LIN {X 0,Y 524.01,Z 370.549,A -85,B 0,C 180,E1 -4760.348,E2 -4760.348} C_VEL
LIN {X 0,Y 523.819,Z 378.444,A -85,B 0,C 180,E1 -4761.318,E2 -4761.318} C_VEL
LIN {X 0,Y 523.619,Z 386.151,A -85,B 0,C 180,E1 -4762.48,E2 -4762.48} C_VEL
LIN {X 0,Y 523.489,Z 393.247,A -85,B 0,C 180,E1 -4763.834,E2 -4763.834} C_VEL
LIN {X 0,Y 523.384,Z 397.968,A -85,B 0,C 180,E1 -4764.992,E2 -4764.992} C_VEL
LIN {X 0,Y 523.444,Z 401.575,A -85,B 0,C 180,E1 -4766.15,E2 -4766.15} C_VEL
LIN {X 0,Y 523.368,Z 403.434,A -85,B 0,C 180,E1 -4766.92,E2 -4766.92} C_VEL
LIN {X 0,Y 523.335,Z 404.828,A -85,B 0,C 180,E1 -4767.69,E2 -4767.69} C_VEL
LIN {X 0,Y 523.251,Z 406.428,A -85,B 0,C 180,E1 -4769.23,E2 -4769.23} C_VEL
LIN {X 0,Y 523.248,Z 406.644,A -85,B 0,C 180,E1 -4769.999,E2 -4769.999} C_VEL
LIN {X 0,Y 523.275,Z 405.822,A -85,B 0,C 180,E1 -4771.538,E2 -4771.538} C_VEL
LIN {X 0,Y 523.335,Z 404.828,A -85,B 0,C 180,E1 -4772.308,E2 -4772.308} C_VEL
LIN {X 0,Y 523.367,Z 403.433,A -85,B 0,C 180,E1 -4773.078,E2 -4773.078} C_VEL
LIN {X 0,Y 523.423,Z 400.501,A -85,B 0,C 180,E1 -4774.234,E2 -4774.234} C_VEL
LIN {X 0,Y 523.461,Z 396.528,A -85,B 0,C 180,E1 -4775.392,E2 -4775.392} C_VEL
LIN {X 0,Y 523.516,Z 391.306,A -85,B 0,C 180,E1 -4776.573,E2 -4776.573} C_VEL
LIN {X 0,Y 523.632,Z 384.971,A -85,B 0,C 180,E1 -4777.712,E2 -4777.712} C_VEL
LIN {X 0,Y 523.81,Z 376.935,A -85,B 0,C 180,E1 -4778.875,E2 -4778.875} C_VEL
LIN {X 0,Y 524.018,Z 368.739,A -85,B 0,C 180,E1 -4779.845,E2 -4779.845} C_VEL
LIN {X 0,Y 524.334,Z 358.741,A -85,B 0,C 180,E1 -4780.815,E2 -4780.815} C_VEL
LIN {X 0,Y 524.628,Z 347.427,A -85,B 0,C 180,E1 -4781.689,E2 -4781.689} C_VEL
LIN {X 0,Y 524.878,Z 336.346,A -85,B 0,C 180,E1 -4782.37,E2 -4782.37} C_VEL
LIN {X 0,Y 525.142,Z 324.039,A -85,B 0,C 180,E1 -4782.953,E2 -4782.953} C_VEL
LIN {X 0,Y 525.376,Z 311.005,A -85,B 0,C 180,E1 -4783.39,E2 -4783.39} C_VEL
LIN {X 0,Y 525.558,Z 298.573,A -85,B 0,C 180,E1 -4783.656,E2 -4783.656} C_VEL
LIN {X 0,Y 525.847,Z 204.835,A -85,B 0,C 180,E1 -4784.959,E2 -4784.959} C_VEL
LIN {X 0,Y 524.268,Z 194.811,A -85,B 0,C 180,E1 -4785.162,E2 -4785.162} C_VEL
LIN {X 0,Y 524.289,Z 192.055,A -85,B 0,C 180,E1 -4785.55,E2 -4785.55} C_VEL
LIN {X 0,Y 524.689,Z 173.78,A -85,B 0,C 180,E1 -4788.528,E2 -4788.528} C_VEL
LIN {X 0,Y 525.146,Z 153.996,A -85,B 0,C 180,E1 -4791.799,E2 -4791.799} C_VEL
LIN {X 0,Y 524.744,Z 149.225,A -85,B 0,C 180,E1 -4792.618,E2 -4792.618} C_VEL
LIN {X 0,Y 523.947,Z 144.887,A -85,B 0,C 180,E1 -4793.413,E2 -4793.413} C_VEL
LIN {X 0,Y 523.895,Z 144.725,A -85,B 0,C 180,E1 -4796.274,E2 -4796.274} C_VEL
LIN {X 0,Y 523.867,Z 144.728,A -85,B 0,C 180,E1 -4798.878,E2 -4798.878} C_VEL
LIN {X 0,Y 523.903,Z 144.728,A -85,B 0,C 180,E1 -4801.544,E2 -4801.544} C_VEL
LIN {X 0,Y 523.906,Z 144.722,A -85,B 0,C 180,E1 -4804.291,E2 -4804.291} C_VEL
LIN {X 0,Y 523.861,Z 144.732,A -85,B 0,C 180,E1 -4807.671,E2 -4807.671} C_VEL
LIN {X 0,Y 523.906,Z 144.721,A -85,B 0,C 180,E1 -4810.125,E2 -4810.125} C_VEL
LIN {X 0,Y 523.864,Z 144.732,A -85,B 0,C 180,E1 -4813.171,E2 -4813.171} C_VEL
LIN {X 0,Y 523.909,Z 144.723,A -85,B 0,C 180,E1 -4815.768,E2 -4815.768} C_VEL
LIN {X 0,Y 523.882,Z 144.728,A -85,B 0,C 180,E1 -4818.902,E2 -4818.902} C_VEL
LIN {X 0,Y 523.891,Z 144.722,A -85,B 0,C 180,E1 -4821.896,E2 -4821.896} C_VEL
LIN {X 0,Y 523.907,Z 144.726,A -85,B 0,C 180,E1 -4824.911,E2 -4824.911} C_VEL
LIN {X 0,Y 523.889,Z 144.724,A -85,B 0,C 180,E1 -4827.685,E2 -4827.685} C_VEL
LIN {X 0,Y 523.919,Z 144.722,A -85,B 0,C 180,E1 -4830.68,E2 -4830.68} C_VEL
LIN {X 0,Y 523.888,Z 144.723,A -85,B 0,C 180,E1 -4833.724,E2 -4833.724} C_VEL
LIN {X 0,Y 523.894,Z 144.722,A -85,B 0,C 180,E1 -4836.268,E2 -4836.268} C_VEL
LIN {X 0,Y 523.929,Z 144.724,A -85,B 0,C 180,E1 -4838.766,E2 -4838.766} C_VEL
LIN {X 0,Y 523.918,Z 144.722,A -85,B 0,C 180,E1 -4841.219,E2 -4841.219} C_VEL
LIN {X 0,Y 523.894,Z 144.721,A -85,B 0,C 180,E1 -4843.637,E2 -4843.637} C_VEL
LIN {X 0,Y 523.897,Z 144.721,A -85,B 0,C 180,E1 -4846.026,E2 -4846.026} C_VEL
LIN {X 0,Y 524,Z 144.712,A -85,B 0,C 180,E1 -4848.393,E2 -4848.393} C_VEL
LIN {X 0,Y 523.967,Z 144.713,A -85,B 0,C 180,E1 -4851.515,E2 -4851.515} C_VEL
LIN {X 0,Y 523.999,Z 144.708,A -85,B 0,C 180,E1 -4853.84,E2 -4853.84} C_VEL
LIN {X 0,Y 524.02,Z 144.71,A -85,B 0,C 180,E1 -4856.924,E2 -4856.924} C_VEL
LIN {X 0,Y 523.982,Z 144.718,A -85,B 0,C 180,E1 -4858.462,E2 -4858.462} C_VEL
LIN {X 0,Y 524.105,Z 144.702,A -85,B 0,C 180,E1 -4860.768,E2 -4860.768} C_VEL
LIN {X 0,Y 524.011,Z 144.707,A -85,B 0,C 180,E1 -4863.075,E2 -4863.075} C_VEL
LIN {X 0,Y 523.998,Z 144.714,A -85,B 0,C 180,E1 -4866.159,E2 -4866.159} C_VEL
LIN {X 0,Y 523.959,Z 144.713,A -85,B 0,C 180,E1 -4869.262,E2 -4869.262} C_VEL
LIN {X 0,Y 523.937,Z 144.725,A -85,B 0,C 180,E1 -4872.393,E2 -4872.393} C_VEL
LIN {X 0,Y 523.907,Z 144.721,A -85,B 0,C 180,E1 -4875.562,E2 -4875.562} C_VEL
LIN {X 0,Y 523.9,Z 144.727,A -85,B 0,C 180,E1 -4877.971,E2 -4877.971} C_VEL
LIN {X 0,Y 523.957,Z 144.721,A -85,B 0,C 180,E1 -4880.41,E2 -4880.41} C_VEL
LIN {X 0,Y 523.894,Z 144.724,A -85,B 0,C 180,E1 -4882.894,E2 -4882.894} C_VEL
LIN {X 0,Y 523.883,Z 144.724,A -85,B 0,C 180,E1 -4885.422,E2 -4885.422} C_VEL
LIN {X 0,Y 523.882,Z 144.732,A -85,B 0,C 180,E1 -4888.004,E2 -4888.004} C_VEL
LIN {X 0,Y 523.917,Z 144.724,A -85,B 0,C 180,E1 -4890.852,E2 -4890.852} C_VEL
LIN {X 0,Y 523.983,Z 144.932,A -85,B 0,C 180,E1 -4892.759,E2 -4892.759} C_VEL
LIN {X 0,Y 524.746,Z 150.857,A -85,B 0,C 180,E1 -4893.865,E2 -4893.865} C_VEL
LIN {X 0,Y 524.446,Z 167.206,A -85,B 0,C 180,E1 -4896.753,E2 -4896.753} C_VEL
LIN {X 0,Y 524.249,Z 179.439,A -85,B 0,C 180,E1 -4898.871,E2 -4898.871} C_VEL
LIN {X 0,Y 525.481,Z 186.461,A -85,B 0,C 180,E1 -4899.038,E2 -4899.038} C_VEL
LIN {X 0,Y 525.936,Z 190.572,A -85,B 0,C 180,E1 -4899.109,E2 -4899.109} C_VEL
LIN {X 0,Y 525.754,Z 232.261,A -85,B 0,C 180,E1 -4899.688,E2 -4899.688} C_VEL
LIN {X 0,Y 524.994,Z 238.101,A -85,B 0,C 180,E1 -4899.748,E2 -4899.748} C_VEL
LIN {X 0,Y 519.456,Z 257.107,A -85,B 0,C 180,E1 -4899.861,E2 -4899.861} C_VEL
LIN {X 0,Y 518.757,Z 262.947,A -85,B 0,C 180,E1 -4899.924,E2 -4899.924} C_VEL
LIN {X 0,Y 518.573,Z 288.396,A -85,B 0,C 180,E1 -4900.31,E2 -4900.31} C_VEL
LIN {X 0,Y 518.38,Z 301.986,A -85,B 0,C 180,E1 -4900.685,E2 -4900.685} C_VEL
LIN {X 0,Y 518.137,Z 314.524,A -85,B 0,C 180,E1 -4901.2,E2 -4901.2} C_VEL
LIN {X 0,Y 517.792,Z 326.753,A -85,B 0,C 180,E1 -4901.876,E2 -4901.876} C_VEL
LIN {X 0,Y 517.482,Z 338.316,A -85,B 0,C 180,E1 -4902.703,E2 -4902.703} C_VEL
LIN {X 0,Y 517.193,Z 348.83,A -85,B 0,C 180,E1 -4903.65,E2 -4903.65} C_VEL
LIN {X 0,Y 516.919,Z 358.553,A -85,B 0,C 180,E1 -4904.736,E2 -4904.736} C_VEL
LIN {X 0,Y 516.679,Z 366.293,A -85,B 0,C 180,E1 -4905.806,E2 -4905.806} C_VEL
LIN {X 0,Y 516.532,Z 372.681,A -85,B 0,C 180,E1 -4906.883,E2 -4906.883} C_VEL
LIN {X 0,Y 516.407,Z 378.822,A -85,B 0,C 180,E1 -4908.177,E2 -4908.177} C_VEL
LIN {X 0,Y 516.331,Z 384.126,A -85,B 0,C 180,E1 -4909.661,E2 -4909.661} C_VEL
LIN {X 0,Y 516.176,Z 387.85,A -85,B 0,C 180,E1 -4911.223,E2 -4911.223} C_VEL
LIN {X 0,Y 516.139,Z 389.373,A -85,B 0,C 180,E1 -4912.214,E2 -4912.214} C_VEL
LIN {X 0,Y 516.127,Z 390.348,A -85,B 0,C 180,E1 -4913.455,E2 -4913.455} C_VEL
LIN {X 0,Y 516.161,Z 390.29,A -85,B 0,C 180,E1 -4914.78,E2 -4914.78} C_VEL
LIN {X 0,Y 516.171,Z 389.02,A -85,B 0,C 180,E1 -4916.155,E2 -4916.155} C_VEL
LIN {X 0,Y 516.28,Z 386.4,A -85,B 0,C 180,E1 -4917.563,E2 -4917.563} C_VEL
LIN {X 0,Y 516.323,Z 382.764,A -85,B 0,C 180,E1 -4918.854,E2 -4918.854} C_VEL
LIN {X 0,Y 516.43,Z 377.59,A -85,B 0,C 180,E1 -4920.195,E2 -4920.195} C_VEL
LIN {X 0,Y 516.542,Z 371.937,A -85,B 0,C 180,E1 -4921.342,E2 -4921.342} C_VEL
LIN {X 0,Y 516.768,Z 363.589,A -85,B 0,C 180,E1 -4922.679,E2 -4922.679} C_VEL
LIN {X 0,Y 517.007,Z 354.868,A -85,B 0,C 180,E1 -4923.789,E2 -4923.789} C_VEL
LIN {X 0,Y 517.288,Z 345.382,A -85,B 0,C 180,E1 -4924.77,E2 -4924.77} C_VEL
LIN {X 0,Y 517.613,Z 334.613,A -85,B 0,C 180,E1 -4925.671,E2 -4925.671} C_VEL
LIN {X 0,Y 517.889,Z 323.665,A -85,B 0,C 180,E1 -4926.403,E2 -4926.403} C_VEL
LIN {X 0,Y 518.19,Z 311.591,A -85,B 0,C 180,E1 -4927.023,E2 -4927.023} C_VEL
LIN {X 0,Y 518.39,Z 298.873,A -85,B 0,C 180,E1 -4927.507,E2 -4927.507} C_VEL
LIN {X 0,Y 518.613,Z 285.867,A -85,B 0,C 180,E1 -4927.833,E2 -4927.833} C_VEL
LIN {X 0,Y 519.067,Z 189.85,A -85,B 0,C 180,E1 -4929.195,E2 -4929.195} C_VEL
LIN {X 0,Y 517.279,Z 179.688,A -85,B 0,C 180,E1 -4929.42,E2 -4929.42} C_VEL
LIN {X 0,Y 517.451,Z 169.81,A -85,B 0,C 180,E1 -4931.183,E2 -4931.183} C_VEL
LIN {X 0,Y 517.932,Z 153.223,A -85,B 0,C 180,E1 -4934.254,E2 -4934.254} C_VEL
LIN {X 0,Y 517.574,Z 149.071,A -85,B 0,C 180,E1 -4935.05,E2 -4935.05} C_VEL
LIN {X 0,Y 516.951,Z 145.624,A -85,B 0,C 180,E1 -4935.786,E2 -4935.786} C_VEL
LIN {X 0,Y 516.948,Z 145.59,A -85,B 0,C 180,E1 -4939.029,E2 -4939.029} C_VEL
LIN {X 0,Y 516.975,Z 145.588,A -85,B 0,C 180,E1 -4942.188,E2 -4942.188} C_VEL
LIN {X 0,Y 517.026,Z 145.578,A -85,B 0,C 180,E1 -4944.541,E2 -4944.541} C_VEL
LIN {X 0,Y 517.08,Z 145.577,A -85,B 0,C 180,E1 -4947.664,E2 -4947.664} C_VEL
LIN {X 0,Y 517.091,Z 145.569,A -85,B 0,C 180,E1 -4950.78,E2 -4950.78} C_VEL
LIN {X 0,Y 517.01,Z 145.581,A -85,B 0,C 180,E1 -4953.118,E2 -4953.118} C_VEL
LIN {X 0,Y 517,Z 145.581,A -85,B 0,C 180,E1 -4956.244,E2 -4956.244} C_VEL
LIN {X 0,Y 516.946,Z 145.594,A -85,B 0,C 180,E1 -4959.39,E2 -4959.39} C_VEL
LIN {X 0,Y 516.95,Z 145.591,A -85,B 0,C 180,E1 -4961.808,E2 -4961.808} C_VEL
LIN {X 0,Y 516.943,Z 145.592,A -85,B 0,C 180,E1 -4965.147,E2 -4965.147} C_VEL
LIN {X 0,Y 516.915,Z 145.591,A -85,B 0,C 180,E1 -4968.223,E2 -4968.223} C_VEL
LIN {X 0,Y 516.911,Z 145.593,A -85,B 0,C 180,E1 -4970.702,E2 -4970.702} C_VEL
LIN {X 0,Y 516.889,Z 145.594,A -85,B 0,C 180,E1 -4974.074,E2 -4974.074} C_VEL
LIN {X 0,Y 516.923,Z 145.592,A -85,B 0,C 180,E1 -4976.658,E2 -4976.658} C_VEL
LIN {X 0,Y 516.908,Z 145.595,A -85,B 0,C 180,E1 -4979.524,E2 -4979.524} C_VEL
LIN {X 0,Y 516.893,Z 145.596,A -85,B 0,C 180,E1 -4982.543,E2 -4982.543} C_VEL
LIN {X 0,Y 516.864,Z 145.601,A -85,B 0,C 180,E1 -4985.33,E2 -4985.33} C_VEL
LIN {X 0,Y 516.878,Z 145.595,A -85,B 0,C 180,E1 -4987.943,E2 -4987.943} C_VEL
LIN {X 0,Y 516.882,Z 145.602,A -85,B 0,C 180,E1 -4990.742,E2 -4990.742} C_VEL
LIN {X 0,Y 516.881,Z 145.604,A -85,B 0,C 180,E1 -4992.832,E2 -4992.832} C_VEL
LIN {X 0,Y 516.894,Z 145.599,A -85,B 0,C 180,E1 -4995.007,E2 -4995.007} C_VEL
LIN {X 0,Y 516.908,Z 145.596,A -85,B 0,C 180,E1 -4998.4,E2 -4998.4} C_VEL
LIN {X 0,Y 516.877,Z 145.596,A -85,B 0,C 180,E1 -5001.284,E2 -5001.284} C_VEL
LIN {X 0,Y 516.866,Z 145.601,A -85,B 0,C 180,E1 -5004.22,E2 -5004.22} C_VEL
LIN {X 0,Y 516.893,Z 145.595,A -85,B 0,C 180,E1 -5007.053,E2 -5007.053} C_VEL
LIN {X 0,Y 516.886,Z 145.596,A -85,B 0,C 180,E1 -5009.796,E2 -5009.796} C_VEL
LIN {X 0,Y 516.891,Z 145.602,A -85,B 0,C 180,E1 -5012.466,E2 -5012.466} C_VEL
LIN {X 0,Y 516.864,Z 145.598,A -85,B 0,C 180,E1 -5015.07,E2 -5015.07} C_VEL
LIN {X 0,Y 516.868,Z 145.598,A -85,B 0,C 180,E1 -5017.622,E2 -5017.622} C_VEL
LIN {X 0,Y 516.928,Z 145.597,A -85,B 0,C 180,E1 -5020.13,E2 -5020.13} C_VEL
LIN {X 0,Y 516.892,Z 145.597,A -85,B 0,C 180,E1 -5022.595,E2 -5022.595} C_VEL
LIN {X 0,Y 516.934,Z 145.588,A -85,B 0,C 180,E1 -5025.03,E2 -5025.03} C_VEL
LIN {X 0,Y 516.966,Z 145.59,A -85,B 0,C 180,E1 -5028.234,E2 -5028.234} C_VEL
LIN {X 0,Y 516.934,Z 145.59,A -85,B 0,C 180,E1 -5031.399,E2 -5031.399} C_VEL
LIN {X 0,Y 516.985,Z 145.583,A -85,B 0,C 180,E1 -5034.54,E2 -5034.54} C_VEL
LIN {X 0,Y 517.072,Z 145.578,A -85,B 0,C 180,E1 -5037.663,E2 -5037.663} C_VEL
LIN {X 0,Y 517.063,Z 145.578,A -85,B 0,C 180,E1 -5040,E2 -5040} C_VEL
LIN {X 0,Y 517.073,Z 145.572,A -85,B 0,C 180,E1 -5042.337,E2 -5042.337} C_VEL
LIN {X 0,Y 516.98,Z 145.589,A -85,B 0,C 180,E1 -5045.461,E2 -5045.461} C_VEL
LIN {X 0,Y 516.926,Z 145.589,A -85,B 0,C 180,E1 -5048.601,E2 -5048.601} C_VEL
LIN {X 0,Y 516.953,Z 145.591,A -85,B 0,C 180,E1 -5051.807,E2 -5051.807} C_VEL
LIN {X 0,Y 516.935,Z 145.593,A -85,B 0,C 180,E1 -5055.142,E2 -5055.142} C_VEL
LIN {X 0,Y 516.876,Z 145.596,A -85,B 0,C 180,E1 -5058.224,E2 -5058.224} C_VEL
LIN {X 0,Y 516.894,Z 145.595,A -85,B 0,C 180,E1 -5060.703,E2 -5060.703} C_VEL
LIN {X 0,Y 516.856,Z 145.606,A -85,B 0,C 180,E1 -5063.225,E2 -5063.225} C_VEL
LIN {X 0,Y 516.86,Z 145.598,A -85,B 0,C 180,E1 -5066.177,E2 -5066.177} C_VEL
LIN {X 0,Y 516.829,Z 145.602,A -85,B 0,C 180,E1 -5068.421,E2 -5068.421} C_VEL
LIN {X 0,Y 516.849,Z 145.608,A -85,B 0,C 180,E1 -5071.113,E2 -5071.113} C_VEL
LIN {X 0,Y 516.871,Z 145.596,A -85,B 0,C 180,E1 -5073.96,E2 -5073.96} C_VEL
LIN {X 0,Y 516.81,Z 145.609,A -85,B 0,C 180,E1 -5076.752,E2 -5076.752} C_VEL
LIN {X 0,Y 516.866,Z 145.602,A -85,B 0,C 180,E1 -5079.19,E2 -5079.19} C_VEL
LIN {X 0,Y 516.832,Z 145.601,A -85,B 0,C 180,E1 -5081.784,E2 -5081.784} C_VEL
LIN {X 0,Y 516.898,Z 145.599,A -85,B 0,C 180,E1 -5085.007,E2 -5085.007} C_VEL
LIN {X 0,Y 516.831,Z 145.605,A -85,B 0,C 180,E1 -5088.41,E2 -5088.41} C_VEL
LIN {X 0,Y 516.85,Z 145.6,A -85,B 0,C 180,E1 -5091.281,E2 -5091.281} C_VEL
LIN {X 0,Y 516.809,Z 145.612,A -85,B 0,C 180,E1 -5094.68,E2 -5094.68} C_VEL
LIN {X 0,Y 516.865,Z 145.597,A -85,B 0,C 180,E1 -5097.463,E2 -5097.463} C_VEL
LIN {X 0,Y 516.84,Z 145.609,A -85,B 0,C 180,E1 -5100.491,E2 -5100.491} C_VEL
LIN {X 0,Y 516.831,Z 145.602,A -85,B 0,C 180,E1 -5103.337,E2 -5103.337} C_VEL
LIN {X 0,Y 516.911,Z 145.72,A -85,B 0,C 180,E1 -5106.3,E2 -5106.3} C_VEL
LIN {X 0,Y 518.219,Z 153.145,A -85,B 0,C 180,E1 -5107.682,E2 -5107.682} C_VEL
LIN {X 0,Y 517.907,Z 166.623,A -85,B 0,C 180,E1 -5109.977,E2 -5109.977} C_VEL
LIN {X 0,Y 517.502,Z 183.566,A -85,B 0,C 180,E1 -5112.819,E2 -5112.819} C_VEL
LIN {X 0,Y 517.266,Z 194.642,A -85,B 0,C 180,E1 -5114.617,E2 -5114.617} C_VEL
LIN {X 0,Y 519.088,Z 206.76,A -85,B 0,C 180,E1 -5114.869,E2 -5114.869} C_VEL
LIN {X 0,Y 518.62,Z 302.588,A -85,B 0,C 180,E1 -5116.231,E2 -5116.231} C_VEL
LIN {X 0,Y 518.394,Z 315.759,A -85,B 0,C 180,E1 -5116.575,E2 -5116.575} C_VEL
LIN {X 0,Y 518.099,Z 328.438,A -85,B 0,C 180,E1 -5117.066,E2 -5117.066} C_VEL
LIN {X 0,Y 517.853,Z 339.954,A -85,B 0,C 180,E1 -5117.672,E2 -5117.672} C_VEL
LIN {X 0,Y 517.56,Z 351.366,A -85,B 0,C 180,E1 -5118.445,E2 -5118.445} C_VEL
LIN {X 0,Y 517.223,Z 361.847,A -85,B 0,C 180,E1 -5119.33,E2 -5119.33} C_VEL
LIN {X 0,Y 516.955,Z 370.414,A -85,B 0,C 180,E1 -5120.215,E2 -5120.215} C_VEL
LIN {X 0,Y 516.756,Z 378.314,A -85,B 0,C 180,E1 -5121.198,E2 -5121.198} C_VEL
LIN {X 0,Y 516.545,Z 386.028,A -85,B 0,C 180,E1 -5122.376,E2 -5122.376} C_VEL
LIN {X 0,Y 516.399,Z 393.129,A -85,B 0,C 180,E1 -5123.749,E2 -5123.749} C_VEL
LIN {X 0,Y 516.313,Z 397.852,A -85,B 0,C 180,E1 -5124.923,E2 -5124.923} C_VEL
LIN {X 0,Y 516.352,Z 401.462,A -85,B 0,C 180,E1 -5126.097,E2 -5126.097} C_VEL
LIN {X 0,Y 516.283,Z 403.323,A -85,B 0,C 180,E1 -5126.878,E2 -5126.878} C_VEL
LIN {X 0,Y 516.262,Z 404.718,A -85,B 0,C 180,E1 -5127.659,E2 -5127.659} C_VEL
LIN {X 0,Y 516.16,Z 406.318,A -85,B 0,C 180,E1 -5129.219,E2 -5129.219} C_VEL
LIN {X 0,Y 516.156,Z 406.534,A -85,B 0,C 180,E1 -5129.999,E2 -5129.999} C_VEL
LIN {X 0,Y 516.192,Z 405.711,A -85,B 0,C 180,E1 -5131.56,E2 -5131.56} C_VEL
LIN {X 0,Y 516.261,Z 404.716,A -85,B 0,C 180,E1 -5132.34,E2 -5132.34} C_VEL
LIN {X 0,Y 516.282,Z 403.319,A -85,B 0,C 180,E1 -5133.12,E2 -5133.12} C_VEL
LIN {X 0,Y 516.311,Z 400.383,A -85,B 0,C 180,E1 -5134.293,E2 -5134.293} C_VEL
LIN {X 0,Y 516.397,Z 396.408,A -85,B 0,C 180,E1 -5135.466,E2 -5135.466} C_VEL
LIN {X 0,Y 516.48,Z 390.481,A -85,B 0,C 180,E1 -5136.8,E2 -5136.8} C_VEL
LIN {X 0,Y 516.586,Z 383.604,A -85,B 0,C 180,E1 -5138.015,E2 -5138.015} C_VEL
LIN {X 0,Y 516.806,Z 375.304,A -85,B 0,C 180,E1 -5139.194,E2 -5139.194} C_VEL
LIN {X 0,Y 517.027,Z 366.785,A -85,B 0,C 180,E1 -5140.177,E2 -5140.177} C_VEL
LIN {X 0,Y 517.375,Z 356.259,A -85,B 0,C 180,E1 -5141.16,E2 -5141.16} C_VEL
LIN {X 0,Y 517.707,Z 344.792,A -85,B 0,C 180,E1 -5142.019,E2 -5142.019} C_VEL
LIN {X 0,Y 517.987,Z 334.391,A -85,B 0,C 180,E1 -5142.636,E2 -5142.636} C_VEL
LIN {X 0,Y 518.243,Z 322.571,A -85,B 0,C 180,E1 -5143.178,E2 -5143.178} C_VEL
LIN {X 0,Y 518.494,Z 308.936,A -85,B 0,C 180,E1 -5143.621,E2 -5143.621} C_VEL
LIN {X 0,Y 518.668,Z 295.053,A -85,B 0,C 180,E1 -5143.891,E2 -5143.891} C_VEL
LIN {X 0,Y 518.972,Z 205.308,A -85,B 0,C 180,E1 -5145.153,E2 -5145.153} C_VEL
LIN {X 0,Y 517.263,Z 194.623,A -85,B 0,C 180,E1 -5145.375,E2 -5145.375} C_VEL
LIN {X 0,Y 517.4,Z 187.023,A -85,B 0,C 180,E1 -5146.573,E2 -5146.573} C_VEL
LIN {X 0,Y 517.776,Z 169.838,A -85,B 0,C 180,E1 -5149.422,E2 -5149.422} C_VEL
LIN {X 0,Y 518.209,Z 153.859,A -85,B 0,C 180,E1 -5152.106,E2 -5152.106} C_VEL
LIN {X 0,Y 516.916,Z 145.723,A -85,B 0,C 180,E1 -5153.591,E2 -5153.591} C_VEL
LIN {X 0,Y 516.833,Z 145.604,A -85,B 0,C 180,E1 -5156.662,E2 -5156.662} C_VEL
LIN {X 0,Y 516.834,Z 145.608,A -85,B 0,C 180,E1 -5159.508,E2 -5159.508} C_VEL
LIN {X 0,Y 516.887,Z 145.596,A -85,B 0,C 180,E1 -5162.541,E2 -5162.541} C_VEL
LIN {X 0,Y 516.844,Z 145.608,A -85,B 0,C 180,E1 -5165.326,E2 -5165.326} C_VEL
LIN {X 0,Y 516.851,Z 145.6,A -85,B 0,C 180,E1 -5168.717,E2 -5168.717} C_VEL
LIN {X 0,Y 516.834,Z 145.605,A -85,B 0,C 180,E1 -5171.781,E2 -5171.781} C_VEL
LIN {X 0,Y 516.888,Z 145.599,A -85,B 0,C 180,E1 -5175.006,E2 -5175.006} C_VEL
LIN {X 0,Y 516.841,Z 145.601,A -85,B 0,C 180,E1 -5178.406,E2 -5178.406} C_VEL
LIN {X 0,Y 516.861,Z 145.605,A -85,B 0,C 180,E1 -5181.282,E2 -5181.282} C_VEL
LIN {X 0,Y 516.849,Z 145.602,A -85,B 0,C 180,E1 -5184.67,E2 -5184.67} C_VEL
LIN {X 0,Y 516.856,Z 145.602,A -85,B 0,C 180,E1 -5187.461,E2 -5187.461} C_VEL
LIN {X 0,Y 516.887,Z 145.598,A -85,B 0,C 180,E1 -5190.693,E2 -5190.693} C_VEL
LIN {X 0,Y 516.868,Z 145.597,A -85,B 0,C 180,E1 -5193.817,E2 -5193.817} C_VEL
LIN {X 0,Y 516.843,Z 145.605,A -85,B 0,C 180,E1 -5196.775,E2 -5196.775} C_VEL
LIN {X 0,Y 516.917,Z 145.59,A -85,B 0,C 180,E1 -5199.734,E2 -5199.734} C_VEL
LIN {X 0,Y 516.88,Z 145.6,A -85,B 0,C 180,E1 -5202.594,E2 -5202.594} C_VEL
LIN {X 0,Y 516.916,Z 145.596,A -85,B 0,C 180,E1 -5205.029,E2 -5205.029} C_VEL
LIN {X 0,Y 516.953,Z 145.588,A -85,B 0,C 180,E1 -5208.233,E2 -5208.233} C_VEL
LIN {X 0,Y 516.935,Z 145.589,A -85,B 0,C 180,E1 -5211.399,E2 -5211.399} C_VEL
LIN {X 0,Y 516.968,Z 145.584,A -85,B 0,C 180,E1 -5213.756,E2 -5213.756} C_VEL
LIN {X 0,Y 516.963,Z 145.59,A -85,B 0,C 180,E1 -5216.882,E2 -5216.882} C_VEL
LIN {X 0,Y 516.95,Z 145.593,A -85,B 0,C 180,E1 -5218.442,E2 -5218.442} C_VEL
LIN {X 0,Y 517.075,Z 145.577,A -85,B 0,C 180,E1 -5220.778,E2 -5220.778} C_VEL
LIN {X 0,Y 516.952,Z 145.586,A -85,B 0,C 180,E1 -5223.117,E2 -5223.117} C_VEL
LIN {X 0,Y 516.967,Z 145.591,A -85,B 0,C 180,E1 -5226.243,E2 -5226.243} C_VEL
LIN {X 0,Y 516.914,Z 145.591,A -85,B 0,C 180,E1 -5229.39,E2 -5229.39} C_VEL
LIN {X 0,Y 516.889,Z 145.601,A -85,B 0,C 180,E1 -5232.565,E2 -5232.565} C_VEL
LIN {X 0,Y 516.928,Z 145.59,A -85,B 0,C 180,E1 -5235.145,E2 -5235.145} C_VEL
LIN {X 0,Y 516.862,Z 145.606,A -85,B 0,C 180,E1 -5238.224,E2 -5238.224} C_VEL
LIN {X 0,Y 516.897,Z 145.597,A -85,B 0,C 180,E1 -5240.702,E2 -5240.702} C_VEL
LIN {X 0,Y 516.87,Z 145.605,A -85,B 0,C 180,E1 -5244.074,E2 -5244.074} C_VEL
LIN {X 0,Y 516.822,Z 145.606,A -85,B 0,C 180,E1 -5246.663,E2 -5246.663} C_VEL
LIN {X 0,Y 516.87,Z 145.602,A -85,B 0,C 180,E1 -5249.519,E2 -5249.519} C_VEL
LIN {X 0,Y 516.937,Z 145.733,A -85,B 0,C 180,E1 -5252.593,E2 -5252.593} C_VEL
LIN {X 0,Y 517.785,Z 152.112,A -85,B 0,C 180,E1 -5253.814,E2 -5253.814} C_VEL
LIN {X 0,Y 517.435,Z 169.647,A -85,B 0,C 180,E1 -5256.942,E2 -5256.942} C_VEL
LIN {X 0,Y 517.285,Z 179.482,A -85,B 0,C 180,E1 -5258.656,E2 -5258.656} C_VEL
LIN {X 0,Y 518.114,Z 184.368,A -85,B 0,C 180,E1 -5258.788,E2 -5258.788} C_VEL
LIN {X 0,Y 519.099,Z 190.699,A -85,B 0,C 180,E1 -5258.908,E2 -5258.908} C_VEL
LIN {X 0,Y 518.757,Z 262.947,A -85,B 0,C 180,E1 -5259.924,E2 -5259.924} C_VEL
LIN {X 0,Y 518.026,Z 268.8,A -85,B 0,C 180,E1 -5259.982,E2 -5259.982} C_VEL
LIN {X 0,Y 512.332,Z 287.754,A -85,B 0,C 180,E1 -5260.122,E2 -5260.122} C_VEL
LIN {X 0,Y 511.653,Z 293.501,A -85,B 0,C 180,E1 -5260.244,E2 -5260.244} C_VEL
LIN {X 0,Y 511.389,Z 306.53,A -85,B 0,C 180,E1 -5260.67,E2 -5260.67} C_VEL
LIN {X 0,Y 511.121,Z 318.867,A -85,B 0,C 180,E1 -5261.241,E2 -5261.241} C_VEL
LIN {X 0,Y 510.819,Z 330.246,A -85,B 0,C 180,E1 -5261.938,E2 -5261.938} C_VEL
LIN {X 0,Y 510.423,Z 341.048,A -85,B 0,C 180,E1 -5262.77,E2 -5262.77} C_VEL
LIN {X 0,Y 510.143,Z 350.656,A -85,B 0,C 180,E1 -5263.685,E2 -5263.685} C_VEL
LIN {X 0,Y 509.87,Z 359.112,A -85,B 0,C 180,E1 -5264.666,E2 -5264.666} C_VEL
LIN {X 0,Y 509.625,Z 367.176,A -85,B 0,C 180,E1 -5265.816,E2 -5265.816} C_VEL
LIN {X 0,Y 509.456,Z 373.805,A -85,B 0,C 180,E1 -5266.981,E2 -5266.981} C_VEL
LIN {X 0,Y 509.332,Z 379.223,A -85,B 0,C 180,E1 -5268.169,E2 -5268.169} C_VEL
LIN {X 0,Y 509.247,Z 384.12,A -85,B 0,C 180,E1 -5269.563,E2 -5269.563} C_VEL
LIN {X 0,Y 509.148,Z 386.847,A -85,B 0,C 180,E1 -5270.623,E2 -5270.623} C_VEL
LIN {X 0,Y 509.056,Z 389.128,A -85,B 0,C 180,E1 -5271.9,E2 -5271.9} C_VEL
LIN {X 0,Y 509.029,Z 390.362,A -85,B 0,C 180,E1 -5273.205,E2 -5273.205} C_VEL
LIN {X 0,Y 509.047,Z 390.497,A -85,B 0,C 180,E1 -5274.561,E2 -5274.561} C_VEL
LIN {X 0,Y 509.067,Z 389.454,A -85,B 0,C 180,E1 -5275.928,E2 -5275.928} C_VEL
LIN {X 0,Y 509.169,Z 386.907,A -85,B 0,C 180,E1 -5277.433,E2 -5277.433} C_VEL
LIN {X 0,Y 509.228,Z 383.142,A -85,B 0,C 180,E1 -5278.834,E2 -5278.834} C_VEL
LIN {X 0,Y 509.362,Z 377.969,A -85,B 0,C 180,E1 -5280.219,E2 -5280.219} C_VEL
LIN {X 0,Y 509.497,Z 371.257,A -85,B 0,C 180,E1 -5281.582,E2 -5281.582} C_VEL
LIN {X 0,Y 509.725,Z 364.247,A -85,B 0,C 180,E1 -5282.715,E2 -5282.715} C_VEL
LIN {X 0,Y 509.974,Z 355.742,A -85,B 0,C 180,E1 -5283.834,E2 -5283.834} C_VEL
LIN {X 0,Y 510.28,Z 345.716,A -85,B 0,C 180,E1 -5284.895,E2 -5284.895} C_VEL
LIN {X 0,Y 510.639,Z 334.687,A -85,B 0,C 180,E1 -5285.831,E2 -5285.831} C_VEL
LIN {X 0,Y 510.972,Z 323.625,A -85,B 0,C 180,E1 -5286.578,E2 -5286.578} C_VEL
LIN {X 0,Y 511.269,Z 311.047,A -85,B 0,C 180,E1 -5287.229,E2 -5287.229} C_VEL
LIN {X 0,Y 511.571,Z 297.863,A -85,B 0,C 180,E1 -5287.724,E2 -5287.724} C_VEL
LIN {X 0,Y 511.741,Z 285.725,A -85,B 0,C 180,E1 -5288.024,E2 -5288.024} C_VEL
LIN {X 0,Y 512.111,Z 189.928,A -85,B 0,C 180,E1 -5289.405,E2 -5289.405} C_VEL
LIN {X 0,Y 510.291,Z 179.816,A -85,B 0,C 180,E1 -5289.632,E2 -5289.632} C_VEL
LIN {X 0,Y 510.408,Z 173.744,A -85,B 0,C 180,E1 -5290.704,E2 -5290.704} C_VEL
LIN {X 0,Y 510.931,Z 155.967,A -85,B 0,C 180,E1 -5294.033,E2 -5294.033} C_VEL
LIN {X 0,Y 510.67,Z 150.691,A -85,B 0,C 180,E1 -5295.047,E2 -5295.047} C_VEL
LIN {X 0,Y 509.889,Z 146.503,A -85,B 0,C 180,E1 -5295.941,E2 -5295.941} C_VEL
LIN {X 0,Y 509.91,Z 146.467,A -85,B 0,C 180,E1 -5298.875,E2 -5298.875} C_VEL
LIN {X 0,Y 509.949,Z 146.465,A -85,B 0,C 180,E1 -5302.079,E2 -5302.079} C_VEL
LIN {X 0,Y 509.978,Z 146.456,A -85,B 0,C 180,E1 -5304.465,E2 -5304.465} C_VEL
LIN {X 0,Y 510.051,Z 146.452,A -85,B 0,C 180,E1 -5307.632,E2 -5307.632} C_VEL
LIN {X 0,Y 510.061,Z 146.445,A -85,B 0,C 180,E1 -5310.79,E2 -5310.79} C_VEL
LIN {X 0,Y 509.952,Z 146.46,A -85,B 0,C 180,E1 -5313.161,E2 -5313.161} C_VEL
LIN {X 0,Y 509.952,Z 146.459,A -85,B 0,C 180,E1 -5316.331,E2 -5316.331} C_VEL
LIN {X 0,Y 509.888,Z 146.475,A -85,B 0,C 180,E1 -5319.521,E2 -5319.521} C_VEL
LIN {X 0,Y 509.903,Z 146.467,A -85,B 0,C 180,E1 -5321.932,E2 -5321.932} C_VEL
LIN {X 0,Y 509.893,Z 146.472,A -85,B 0,C 180,E1 -5325.242,E2 -5325.242} C_VEL
LIN {X 0,Y 509.86,Z 146.47,A -85,B 0,C 180,E1 -5328.484,E2 -5328.484} C_VEL
LIN {X 0,Y 509.849,Z 146.476,A -85,B 0,C 180,E1 -5331.002,E2 -5331.002} C_VEL
LIN {X 0,Y 509.821,Z 146.479,A -85,B 0,C 180,E1 -5333.564,E2 -5333.564} C_VEL
LIN {X 0,Y 509.91,Z 146.464,A -85,B 0,C 180,E1 -5336.379,E2 -5336.379} C_VEL
LIN {X 0,Y 509.871,Z 146.473,A -85,B 0,C 180,E1 -5338.845,E2 -5338.845} C_VEL
LIN {X 0,Y 509.817,Z 146.477,A -85,B 0,C 180,E1 -5341.591,E2 -5341.591} C_VEL
LIN {X 0,Y 509.837,Z 146.474,A -85,B 0,C 180,E1 -5344.415,E2 -5344.415} C_VEL
LIN {X 0,Y 509.815,Z 146.478,A -85,B 0,C 180,E1 -5347.341,E2 -5347.341} C_VEL
LIN {X 0,Y 509.836,Z 146.475,A -85,B 0,C 180,E1 -5350.383,E2 -5350.383} C_VEL
LIN {X 0,Y 509.821,Z 146.48,A -85,B 0,C 180,E1 -5353.062,E2 -5353.062} C_VEL
LIN {X 0,Y 509.821,Z 146.475,A -85,B 0,C 180,E1 -5355.794,E2 -5355.794} C_VEL
LIN {X 0,Y 509.851,Z 146.478,A -85,B 0,C 180,E1 -5358.575,E2 -5358.575} C_VEL
LIN {X 0,Y 509.848,Z 146.471,A -85,B 0,C 180,E1 -5361.787,E2 -5361.787} C_VEL
LIN {X 0,Y 509.826,Z 146.482,A -85,B 0,C 180,E1 -5364.622,E2 -5364.622} C_VEL
LIN {X 0,Y 509.86,Z 146.47,A -85,B 0,C 180,E1 -5367.481,E2 -5367.481} C_VEL
LIN {X 0,Y 509.857,Z 146.476,A -85,B 0,C 180,E1 -5370.274,E2 -5370.274} C_VEL
LIN {X 0,Y 509.873,Z 146.469,A -85,B 0,C 180,E1 -5373.63,E2 -5373.63} C_VEL
LIN {X 0,Y 509.82,Z 146.481,A -85,B 0,C 180,E1 -5376.436,E2 -5376.436} C_VEL
LIN {X 0,Y 509.914,Z 146.466,A -85,B 0,C 180,E1 -5379.845,E2 -5379.845} C_VEL
LIN {X 0,Y 509.86,Z 146.47,A -85,B 0,C 180,E1 -5383.174,E2 -5383.174} C_VEL
LIN {X 0,Y 509.852,Z 146.473,A -85,B 0,C 180,E1 -5385.634,E2 -5385.634} C_VEL
LIN {X 0,Y 509.91,Z 146.464,A -85,B 0,C 180,E1 -5388.875,E2 -5388.875} C_VEL
LIN {X 0,Y 509.878,Z 146.474,A -85,B 0,C 180,E1 -5392.078,E2 -5392.078} C_VEL
LIN {X 0,Y 509.94,Z 146.461,A -85,B 0,C 180,E1 -5394.464,E2 -5394.464} C_VEL
LIN {X 0,Y 510.04,Z 146.453,A -85,B 0,C 180,E1 -5397.631,E2 -5397.631} C_VEL
LIN {X 0,Y 510.032,Z 146.454,A -85,B 0,C 180,E1 -5400,E2 -5400} C_VEL
LIN {X 0,Y 510.043,Z 146.448,A -85,B 0,C 180,E1 -5402.369,E2 -5402.369} C_VEL
LIN {X 0,Y 509.933,Z 146.468,A -85,B 0,C 180,E1 -5405.537,E2 -5405.537} C_VEL
LIN {X 0,Y 509.877,Z 146.472,A -85,B 0,C 180,E1 -5407.923,E2 -5407.923} C_VEL
LIN {X 0,Y 509.907,Z 146.467,A -85,B 0,C 180,E1 -5411.126,E2 -5411.126} C_VEL
LIN {X 0,Y 509.841,Z 146.472,A -85,B 0,C 180,E1 -5414.367,E2 -5414.367} C_VEL
LIN {X 0,Y 509.82,Z 146.476,A -85,B 0,C 180,E1 -5416.828,E2 -5416.828} C_VEL
LIN {X 0,Y 509.89,Z 146.466,A -85,B 0,C 180,E1 -5420.157,E2 -5420.157} C_VEL
LIN {X 0,Y 509.812,Z 146.48,A -85,B 0,C 180,E1 -5423.565,E2 -5423.565} C_VEL
LIN {X 0,Y 509.8,Z 146.477,A -85,B 0,C 180,E1 -5426.353,E2 -5426.353} C_VEL
LIN {X 0,Y 509.793,Z 146.482,A -85,B 0,C 180,E1 -5428.85,E2 -5428.85} C_VEL
LIN {X 0,Y 509.788,Z 146.481,A -85,B 0,C 180,E1 -5431.593,E2 -5431.593} C_VEL
LIN {X 0,Y 509.829,Z 146.475,A -85,B 0,C 180,E1 -5434.416,E2 -5434.416} C_VEL
LIN {X 0,Y 509.78,Z 146.483,A -85,B 0,C 180,E1 -5437.344,E2 -5437.344} C_VEL
LIN {X 0,Y 509.787,Z 146.481,A -85,B 0,C 180,E1 -5440.388,E2 -5440.388} C_VEL
LIN {X 0,Y 509.792,Z 146.479,A -85,B 0,C 180,E1 -5443.575,E2 -5443.575} C_VEL
LIN {X 0,Y 509.793,Z 146.482,A -85,B 0,C 180,E1 -5446.425,E2 -5446.425} C_VEL
LIN {X 0,Y 509.788,Z 146.479,A -85,B 0,C 180,E1 -5449.613,E2 -5449.613} C_VEL
LIN {X 0,Y 509.758,Z 146.491,A -85,B 0,C 180,E1 -5452.654,E2 -5452.654} C_VEL
LIN {X 0,Y 509.814,Z 146.476,A -85,B 0,C 180,E1 -5455.805,E2 -5455.805} C_VEL
LIN {X 0,Y 509.817,Z 146.482,A -85,B 0,C 180,E1 -5458.726,E2 -5458.726} C_VEL
LIN {X 0,Y 509.824,Z 146.48,A -85,B 0,C 180,E1 -5462.05,E2 -5462.05} C_VEL
LIN {X 0,Y 509.789,Z 146.484,A -85,B 0,C 180,E1 -5464.699,E2 -5464.699} C_VEL
LIN {X 0,Y 509.864,Z 146.571,A -85,B 0,C 180,E1 -5466.114,E2 -5466.114} C_VEL
LIN {X 0,Y 511.247,Z 154.263,A -85,B 0,C 180,E1 -5467.575,E2 -5467.575} C_VEL
LIN {X 0,Y 511.02,Z 165.748,A -85,B 0,C 180,E1 -5469.561,E2 -5469.561} C_VEL
LIN {X 0,Y 510.57,Z 182.247,A -85,B 0,C 180,E1 -5472.372,E2 -5472.372} C_VEL
LIN {X 0,Y 510.273,Z 194.51,A -85,B 0,C 180,E1 -5474.399,E2 -5474.399} C_VEL
LIN {X 0,Y 512.241,Z 206.941,A -85,B 0,C 180,E1 -5474.666,E2 -5474.666} C_VEL
LIN {X 0,Y 511.738,Z 302.343,A -85,B 0,C 180,E1 -5476.042,E2 -5476.042} C_VEL
LIN {X 0,Y 511.482,Z 315.555,A -85,B 0,C 180,E1 -5476.39,E2 -5476.39} C_VEL
LIN {X 0,Y 511.158,Z 328.258,A -85,B 0,C 180,E1 -5476.887,E2 -5476.887} C_VEL
LIN {X 0,Y 510.896,Z 339.874,A -85,B 0,C 180,E1 -5477.507,E2 -5477.507} C_VEL
LIN {X 0,Y 510.589,Z 351.217,A -85,B 0,C 180,E1 -5478.285,E2 -5478.285} C_VEL
LIN {X 0,Y 510.232,Z 361.706,A -85,B 0,C 180,E1 -5479.182,E2 -5479.182} C_VEL
LIN {X 0,Y 509.928,Z 370.279,A -85,B 0,C 180,E1 -5480.079,E2 -5480.079} C_VEL
LIN {X 0,Y 509.69,Z 378.185,A -85,B 0,C 180,E1 -5481.075,E2 -5481.075} C_VEL
LIN {X 0,Y 509.495,Z 385.905,A -85,B 0,C 180,E1 -5482.27,E2 -5482.27} C_VEL
LIN {X 0,Y 509.309,Z 393.01,A -85,B 0,C 180,E1 -5483.661,E2 -5483.661} C_VEL
LIN {X 0,Y 509.247,Z 397.737,A -85,B 0,C 180,E1 -5484.853,E2 -5484.853} C_VEL
LIN {X 0,Y 509.246,Z 401.349,A -85,B 0,C 180,E1 -5486.042,E2 -5486.042} C_VEL
LIN {X 0,Y 509.201,Z 403.211,A -85,B 0,C 180,E1 -5486.834,E2 -5486.834} C_VEL
LIN {X 0,Y 509.162,Z 404.607,A -85,B 0,C 180,E1 -5487.626,E2 -5487.626} C_VEL
LIN {X 0,Y 509.074,Z 406.208,A -85,B 0,C 180,E1 -5489.208,E2 -5489.208} C_VEL
LIN {X 0,Y 509.067,Z 406.424,A -85,B 0,C 180,E1 -5489.999,E2 -5489.999} C_VEL
LIN {X 0,Y 509.113,Z 405.599,A -85,B 0,C 180,E1 -5491.581,E2 -5491.581} C_VEL
LIN {X 0,Y 509.161,Z 404.603,A -85,B 0,C 180,E1 -5492.372,E2 -5492.372} C_VEL
LIN {X 0,Y 509.2,Z 403.205,A -85,B 0,C 180,E1 -5493.164,E2 -5493.164} C_VEL
LIN {X 0,Y 509.204,Z 400.266,A -85,B 0,C 180,E1 -5494.353,E2 -5494.353} C_VEL
LIN {X 0,Y 509.31,Z 396.288,A -85,B 0,C 180,E1 -5495.542,E2 -5495.542} C_VEL
LIN {X 0,Y 509.402,Z 390.619,A -85,B 0,C 180,E1 -5496.843,E2 -5496.843} C_VEL
LIN {X 0,Y 509.537,Z 383.472,A -85,B 0,C 180,E1 -5498.127,E2 -5498.127} C_VEL
LIN {X 0,Y 509.763,Z 375.166,A -85,B 0,C 180,E1 -5499.322,E2 -5499.322} C_VEL
LIN {X 0,Y 510.012,Z 366.639,A -85,B 0,C 180,E1 -5500.319,E2 -5500.319} C_VEL
LIN {X 0,Y 510.375,Z 356.102,A -85,B 0,C 180,E1 -5501.315,E2 -5501.315} C_VEL
LIN {X 0,Y 510.716,Z 345.376,A -85,B 0,C 180,E1 -5502.134,E2 -5502.134} C_VEL
LIN {X 0,Y 511.038,Z 334.21,A -85,B 0,C 180,E1 -5502.811,E2 -5502.811} C_VEL
LIN {X 0,Y 511.317,Z 322.365,A -85,B 0,C 180,E1 -5503.36,E2 -5503.36} C_VEL
LIN {X 0,Y 511.605,Z 308.701,A -85,B 0,C 180,E1 -5503.808,E2 -5503.808} C_VEL
LIN {X 0,Y 511.777,Z 296.459,A -85,B 0,C 180,E1 -5504.056,E2 -5504.056} C_VEL
LIN {X 0,Y 512.155,Z 206.296,A -85,B 0,C 180,E1 -5505.344,E2 -5505.344} C_VEL
LIN {X 0,Y 510.285,Z 194.511,A -85,B 0,C 180,E1 -5505.592,E2 -5505.592} C_VEL
LIN {X 0,Y 510.358,Z 189.377,A -85,B 0,C 180,E1 -5506.396,E2 -5506.396} C_VEL
LIN {X 0,Y 510.747,Z 173.405,A -85,B 0,C 180,E1 -5509.074,E2 -5509.074} C_VEL
LIN {X 0,Y 511.254,Z 156.194,A -85,B 0,C 180,E1 -5511.998,E2 -5511.998} C_VEL
LIN {X 0,Y 510.808,Z 151.644,A -85,B 0,C 180,E1 -5512.805,E2 -5512.805} C_VEL
LIN {X 0,Y 509.85,Z 146.576,A -85,B 0,C 180,E1 -5513.777,E2 -5513.777} C_VEL
LIN {X 0,Y 509.814,Z 146.48,A -85,B 0,C 180,E1 -5517.058,E2 -5517.058} C_VEL
LIN {X 0,Y 509.78,Z 146.488,A -85,B 0,C 180,E1 -5519.755,E2 -5519.755} C_VEL
LIN {X 0,Y 509.839,Z 146.475,A -85,B 0,C 180,E1 -5522.767,E2 -5522.767} C_VEL
LIN {X 0,Y 509.789,Z 146.487,A -85,B 0,C 180,E1 -5525.572,E2 -5525.572} C_VEL
LIN {X 0,Y 509.799,Z 146.478,A -85,B 0,C 180,E1 -5528.341,E2 -5528.341} C_VEL
LIN {X 0,Y 509.793,Z 146.486,A -85,B 0,C 180,E1 -5531.43,E2 -5531.43} C_VEL
LIN {X 0,Y 509.826,Z 146.475,A -85,B 0,C 180,E1 -5534.669,E2 -5534.669} C_VEL
LIN {X 0,Y 509.78,Z 146.486,A -85,B 0,C 180,E1 -5537.504,E2 -5537.504} C_VEL
LIN {X 0,Y 509.82,Z 146.477,A -85,B 0,C 180,E1 -5540.645,E2 -5540.645} C_VEL
LIN {X 0,Y 509.793,Z 146.481,A -85,B 0,C 180,E1 -5543.644,E2 -5543.644} C_VEL
LIN {X 0,Y 509.823,Z 146.475,A -85,B 0,C 180,E1 -5546.536,E2 -5546.536} C_VEL
LIN {X 0,Y 509.793,Z 146.483,A -85,B 0,C 180,E1 -5549.33,E2 -5549.33} C_VEL
LIN {X 0,Y 509.818,Z 146.474,A -85,B 0,C 180,E1 -5552.05,E2 -5552.05} C_VEL
LIN {X 0,Y 509.787,Z 146.484,A -85,B 0,C 180,E1 -5554.699,E2 -5554.699} C_VEL
LIN {X 0,Y 509.812,Z 146.478,A -85,B 0,C 180,E1 -5557.458,E2 -5557.458} C_VEL
LIN {X 0,Y 509.894,Z 146.465,A -85,B 0,C 180,E1 -5559.843,E2 -5559.843} C_VEL
LIN {X 0,Y 509.844,Z 146.475,A -85,B 0,C 180,E1 -5563.173,E2 -5563.173} C_VEL
LIN {X 0,Y 509.829,Z 146.473,A -85,B 0,C 180,E1 -5565.633,E2 -5565.633} C_VEL
LIN {X 0,Y 509.893,Z 146.471,A -85,B 0,C 180,E1 -5568.874,E2 -5568.874} C_VEL
LIN {X 0,Y 509.905,Z 146.465,A -85,B 0,C 180,E1 -5572.077,E2 -5572.077} C_VEL
LIN {X 0,Y 509.948,Z 146.464,A -85,B 0,C 180,E1 -5574.464,E2 -5574.464} C_VEL
LIN {X 0,Y 510.027,Z 146.449,A -85,B 0,C 180,E1 -5577.63,E2 -5577.63} C_VEL
LIN {X 0,Y 510.046,Z 146.453,A -85,B 0,C 180,E1 -5580.789,E2 -5580.789} C_VEL
LIN {X 0,Y 509.894,Z 146.465,A -85,B 0,C 180,E1 -5583.16,E2 -5583.16} C_VEL
LIN {X 0,Y 509.922,Z 146.469,A -85,B 0,C 180,E1 -5586.33,E2 -5586.33} C_VEL
LIN {X 0,Y 509.866,Z 146.473,A -85,B 0,C 180,E1 -5588.721,E2 -5588.721} C_VEL
LIN {X 0,Y 509.885,Z 146.47,A -85,B 0,C 180,E1 -5591.932,E2 -5591.932} C_VEL
LIN {X 0,Y 509.88,Z 146.468,A -85,B 0,C 180,E1 -5595.242,E2 -5595.242} C_VEL
LIN {X 0,Y 509.822,Z 146.481,A -85,B 0,C 180,E1 -5598.485,E2 -5598.485} C_VEL
LIN {X 0,Y 509.835,Z 146.475,A -85,B 0,C 180,E1 -5601.002,E2 -5601.002} C_VEL
LIN {X 0,Y 509.804,Z 146.48,A -85,B 0,C 180,E1 -5603.564,E2 -5603.564} C_VEL
LIN {X 0,Y 509.8,Z 146.483,A -85,B 0,C 180,E1 -5606.357,E2 -5606.357} C_VEL
LIN {X 0,Y 509.818,Z 146.479,A -85,B 0,C 180,E1 -5608.847,E2 -5608.847} C_VEL
LIN {X 0,Y 509.855,Z 146.479,A -85,B 0,C 180,E1 -5612.052,E2 -5612.052} C_VEL
LIN {X 0,Y 509.891,Z 146.641,A -85,B 0,C 180,E1 -5612.458,E2 -5612.458} C_VEL
LIN {X 0,Y 510.817,Z 152.677,A -85,B 0,C 180,E1 -5613.626,E2 -5613.626} C_VEL
LIN {X 0,Y 510.469,Z 169.41,A -85,B 0,C 180,E1 -5616.649,E2 -5616.649} C_VEL
LIN {X 0,Y 510.3,Z 179.573,A -85,B 0,C 180,E1 -5618.439,E2 -5618.439} C_VEL
LIN {X 0,Y 511.436,Z 186.087,A -85,B 0,C 180,E1 -5618.605,E2 -5618.605} C_VEL
LIN {X 0,Y 512.269,Z 192.06,A -85,B 0,C 180,E1 -5618.72,E2 -5618.72} C_VEL
LIN {X 0,Y 511.707,Z 287.651,A -85,B 0,C 180,E1 -5620.106,E2 -5620.106} C_VEL
LIN {X 0,Y 511.653,Z 293.501,A -85,B 0,C 180,E1 -5620.244,E2 -5620.244} C_VEL
LIN {X 0,Y 510.385,Z 301.067,A -85,B 0,C 180,E1 -5620.44,E2 -5620.44} C_VEL
LIN {X 0,Y 507.797,Z 308.366,A -85,B 0,C 180,E1 -5620.646,E2 -5620.646} C_VEL
LIN {X 0,Y 504.846,Z 317.352,A -85,B 0,C 180,E1 -5620.996,E2 -5620.996} C_VEL
LIN {X 0,Y 504.077,Z 322.618,A -85,B 0,C 180,E1 -5621.273,E2 -5621.273} C_VEL
LIN {X 0,Y 503.736,Z 334.126,A -85,B 0,C 180,E1 -5622.042,E2 -5622.042} C_VEL
LIN {X 0,Y 503.4,Z 343.879,A -85,B 0,C 180,E1 -5622.859,E2 -5622.859} C_VEL
LIN {X 0,Y 503.011,Z 354.06,A -85,B 0,C 180,E1 -5623.909,E2 -5623.909} C_VEL
LIN {X 0,Y 502.718,Z 362.984,A -85,B 0,C 180,E1 -5625.047,E2 -5625.047} C_VEL
LIN {X 0,Y 502.498,Z 370.19,A -85,B 0,C 180,E1 -5626.186,E2 -5626.186} C_VEL
LIN {X 0,Y 502.306,Z 377.029,A -85,B 0,C 180,E1 -5627.541,E2 -5627.541} C_VEL
LIN {X 0,Y 502.213,Z 382.251,A -85,B 0,C 180,E1 -5628.876,E2 -5628.876} C_VEL
LIN {X 0,Y 502.069,Z 386.44,A -85,B 0,C 180,E1 -5630.344,E2 -5630.344} C_VEL
LIN {X 0,Y 501.994,Z 388.898,A -85,B 0,C 180,E1 -5631.629,E2 -5631.629} C_VEL
LIN {X 0,Y 501.932,Z 390.345,A -85,B 0,C 180,E1 -5632.983,E2 -5632.983} C_VEL
LIN {X 0,Y 501.961,Z 390.667,A -85,B 0,C 180,E1 -5634.297,E2 -5634.297} C_VEL
LIN {X 0,Y 501.992,Z 389.583,A -85,B 0,C 180,E1 -5635.945,E2 -5635.945} C_VEL
LIN {X 0,Y 502.047,Z 387.73,A -85,B 0,C 180,E1 -5637.131,E2 -5637.131} C_VEL
LIN {X 0,Y 502.16,Z 384.114,A -85,B 0,C 180,E1 -5638.619,E2 -5638.619} C_VEL
LIN {X 0,Y 502.2,Z 380.321,A -85,B 0,C 180,E1 -5639.75,E2 -5639.75} C_VEL
LIN {X 0,Y 502.379,Z 374.198,A -85,B 0,C 180,E1 -5641.144,E2 -5641.144} C_VEL
LIN {X 0,Y 502.582,Z 367.563,A -85,B 0,C 180,E1 -5642.337,E2 -5642.337} C_VEL
LIN {X 0,Y 502.794,Z 359.932,A -85,B 0,C 180,E1 -5643.454,E2 -5643.454} C_VEL
LIN {X 0,Y 503.143,Z 350.566,A -85,B 0,C 180,E1 -5644.564,E2 -5644.564} C_VEL
LIN {X 0,Y 503.524,Z 339.925,A -85,B 0,C 180,E1 -5645.577,E2 -5645.577} C_VEL
LIN {X 0,Y 503.851,Z 329.737,A -85,B 0,C 180,E1 -5646.359,E2 -5646.359} C_VEL
LIN {X 0,Y 504.184,Z 317.855,A -85,B 0,C 180,E1 -5647.082,E2 -5647.082} C_VEL
LIN {X 0,Y 504.472,Z 305.761,A -85,B 0,C 180,E1 -5647.637,E2 -5647.637} C_VEL
LIN {X 0,Y 504.737,Z 292.98,A -85,B 0,C 180,E1 -5648.053,E2 -5648.053} C_VEL
LIN {X 0,Y 504.9,Z 280.65,A -85,B 0,C 180,E1 -5648.302,E2 -5648.302} C_VEL
LIN {X 0,Y 505.274,Z 190.829,A -85,B 0,C 180,E1 -5649.603,E2 -5649.603} C_VEL
LIN {X 0,Y 503.339,Z 180.195,A -85,B 0,C 180,E1 -5649.837,E2 -5649.837} C_VEL
LIN {X 0,Y 503.304,Z 178.879,A -85,B 0,C 180,E1 -5649.996,E2 -5649.996} C_VEL
LIN {X 0,Y 503.718,Z 163.148,A -85,B 0,C 180,E1 -5652.964,E2 -5652.964} C_VEL
LIN {X 0,Y 503.965,Z 154.383,A -85,B 0,C 180,E1 -5654.636,E2 -5654.636} C_VEL
LIN {X 0,Y 502.878,Z 147.483,A -85,B 0,C 180,E1 -5656.051,E2 -5656.051} C_VEL
LIN {X 0,Y 502.874,Z 147.344,A -85,B 0,C 180,E1 -5658.718,E2 -5658.718} C_VEL
LIN {X 0,Y 502.899,Z 147.345,A -85,B 0,C 180,E1 -5661.968,E2 -5661.968} C_VEL
LIN {X 0,Y 502.934,Z 147.334,A -85,B 0,C 180,E1 -5664.387,E2 -5664.387} C_VEL
LIN {X 0,Y 503.021,Z 147.327,A -85,B 0,C 180,E1 -5667.599,E2 -5667.599} C_VEL
LIN {X 0,Y 503.024,Z 147.326,A -85,B 0,C 180,E1 -5670.001,E2 -5670.001} C_VEL
LIN {X 0,Y 503.021,Z 147.322,A -85,B 0,C 180,E1 -5672.403,E2 -5672.403} C_VEL
LIN {X 0,Y 502.93,Z 147.342,A -85,B 0,C 180,E1 -5675.614,E2 -5675.614} C_VEL
LIN {X 0,Y 502.879,Z 147.342,A -85,B 0,C 180,E1 -5678.034,E2 -5678.034} C_VEL
LIN {X 0,Y 502.875,Z 147.345,A -85,B 0,C 180,E1 -5681.284,E2 -5681.284} C_VEL
LIN {X 0,Y 502.843,Z 147.344,A -85,B 0,C 180,E1 -5684.572,E2 -5684.572} C_VEL
LIN {X 0,Y 502.821,Z 147.348,A -85,B 0,C 180,E1 -5687.909,E2 -5687.909} C_VEL
LIN {X 0,Y 502.828,Z 147.346,A -85,B 0,C 180,E1 -5690.537,E2 -5690.537} C_VEL
LIN {X 0,Y 502.787,Z 147.356,A -85,B 0,C 180,E1 -5693.041,E2 -5693.041} C_VEL
LIN {X 0,Y 502.819,Z 147.349,A -85,B 0,C 180,E1 -5695.677,E2 -5695.677} C_VEL
LIN {X 0,Y 502.836,Z 147.345,A -85,B 0,C 180,E1 -5698.373,E2 -5698.373} C_VEL
LIN {X 0,Y 502.791,Z 147.353,A -85,B 0,C 180,E1 -5701.499,E2 -5701.499} C_VEL
LIN {X 0,Y 502.788,Z 147.351,A -85,B 0,C 180,E1 -5703.996,E2 -5703.996} C_VEL
LIN {X 0,Y 502.776,Z 147.357,A -85,B 0,C 180,E1 -5707.178,E2 -5707.178} C_VEL
LIN {X 0,Y 502.784,Z 147.351,A -85,B 0,C 180,E1 -5710.016,E2 -5710.016} C_VEL
LIN {X 0,Y 502.802,Z 147.35,A -85,B 0,C 180,E1 -5712.2,E2 -5712.2} C_VEL
LIN {X 0,Y 502.784,Z 147.352,A -85,B 0,C 180,E1 -5715.471,E2 -5715.471} C_VEL
LIN {X 0,Y 502.793,Z 147.35,A -85,B 0,C 180,E1 -5717.861,E2 -5717.861} C_VEL
LIN {X 0,Y 502.799,Z 147.353,A -85,B 0,C 180,E1 -5721.024,E2 -5721.024} C_VEL
LIN {X 0,Y 502.77,Z 147.356,A -85,B 0,C 180,E1 -5724.17,E2 -5724.17} C_VEL
LIN {X 0,Y 502.832,Z 147.348,A -85,B 0,C 180,E1 -5726.994,E2 -5726.994} C_VEL
LIN {X 0,Y 502.813,Z 147.351,A -85,B 0,C 180,E1 -5730.066,E2 -5730.066} C_VEL
LIN {X 0,Y 502.843,Z 147.344,A -85,B 0,C 180,E1 -5733.444,E2 -5733.444} C_VEL
LIN {X 0,Y 502.772,Z 147.358,A -85,B 0,C 180,E1 -5736.086,E2 -5736.086} C_VEL
LIN {X 0,Y 502.78,Z 147.354,A -85,B 0,C 180,E1 -5738.689,E2 -5738.689} C_VEL
LIN {X 0,Y 502.821,Z 147.347,A -85,B 0,C 180,E1 -5741.248,E2 -5741.248} C_VEL
LIN {X 0,Y 502.848,Z 147.346,A -85,B 0,C 180,E1 -5744.601,E2 -5744.601} C_VEL
LIN {X 0,Y 502.876,Z 147.349,A -85,B 0,C 180,E1 -5748.04,E2 -5748.04} C_VEL
LIN {X 0,Y 502.851,Z 147.343,A -85,B 0,C 180,E1 -5751.157,E2 -5751.157} C_VEL
LIN {X 0,Y 502.869,Z 147.344,A -85,B 0,C 180,E1 -5753.581,E2 -5753.581} C_VEL
LIN {X 0,Y 502.836,Z 147.345,A -85,B 0,C 180,E1 -5756.795,E2 -5756.795} C_VEL
LIN {X 0,Y 502.89,Z 147.339,A -85,B 0,C 180,E1 -5758.399,E2 -5758.399} C_VEL
LIN {X 0,Y 503.001,Z 147.33,A -85,B 0,C 180,E1 -5760,E2 -5760} C_VEL
LIN {X 0,Y 503.013,Z 147.324,A -85,B 0,C 180,E1 -5762.403,E2 -5762.403} C_VEL
LIN {X 0,Y 502.888,Z 147.346,A -85,B 0,C 180,E1 -5765.614,E2 -5765.614} C_VEL
LIN {X 0,Y 502.849,Z 147.346,A -85,B 0,C 180,E1 -5768.035,E2 -5768.035} C_VEL
LIN {X 0,Y 502.873,Z 147.345,A -85,B 0,C 180,E1 -5771.284,E2 -5771.284} C_VEL
LIN {X 0,Y 502.823,Z 147.346,A -85,B 0,C 180,E1 -5774.572,E2 -5774.572} C_VEL
LIN {X 0,Y 502.801,Z 147.351,A -85,B 0,C 180,E1 -5777.91,E2 -5777.91} C_VEL
LIN {X 0,Y 502.831,Z 147.346,A -85,B 0,C 180,E1 -5780.536,E2 -5780.536} C_VEL
LIN {X 0,Y 502.785,Z 147.356,A -85,B 0,C 180,E1 -5783.041,E2 -5783.041} C_VEL
LIN {X 0,Y 502.762,Z 147.357,A -85,B 0,C 180,E1 -5785.68,E2 -5785.68} C_VEL
LIN {X 0,Y 502.76,Z 147.354,A -85,B 0,C 180,E1 -5788.378,E2 -5788.378} C_VEL
LIN {X 0,Y 502.766,Z 147.357,A -85,B 0,C 180,E1 -5791.493,E2 -5791.493} C_VEL
LIN {X 0,Y 502.782,Z 147.353,A -85,B 0,C 180,E1 -5794.44,E2 -5794.44} C_VEL
LIN {X 0,Y 502.734,Z 147.363,A -85,B 0,C 180,E1 -5797.171,E2 -5797.171} C_VEL
LIN {X 0,Y 502.734,Z 147.357,A -85,B 0,C 180,E1 -5800.021,E2 -5800.021} C_VEL
LIN {X 0,Y 502.738,Z 147.36,A -85,B 0,C 180,E1 -5803.235,E2 -5803.235} C_VEL
LIN {X 0,Y 502.768,Z 147.353,A -85,B 0,C 180,E1 -5805.658,E2 -5805.658} C_VEL
LIN {X 0,Y 502.752,Z 147.36,A -85,B 0,C 180,E1 -5809.014,E2 -5809.014} C_VEL
LIN {X 0,Y 502.744,Z 147.357,A -85,B 0,C 180,E1 -5812.041,E2 -5812.041} C_VEL
LIN {X 0,Y 502.759,Z 147.354,A -85,B 0,C 180,E1 -5815.564,E2 -5815.564} C_VEL
LIN {X 0,Y 502.767,Z 147.362,A -85,B 0,C 180,E1 -5818.507,E2 -5818.507} C_VEL
LIN {X 0,Y 502.766,Z 147.357,A -85,B 0,C 180,E1 -5821.722,E2 -5821.722} C_VEL
LIN {X 0,Y 502.764,Z 147.362,A -85,B 0,C 180,E1 -5824.32,E2 -5824.32} C_VEL
LIN {X 0,Y 502.834,Z 147.542,A -85,B 0,C 180,E1 -5825.978,E2 -5825.978} C_VEL
LIN {X 0,Y 504.363,Z 156.596,A -85,B 0,C 180,E1 -5827.684,E2 -5827.684} C_VEL
LIN {X 0,Y 503.894,Z 171.196,A -85,B 0,C 180,E1 -5830.231,E2 -5830.231} C_VEL
LIN {X 0,Y 503.489,Z 185.789,A -85,B 0,C 180,E1 -5832.745,E2 -5832.745} C_VEL
LIN {X 0,Y 503.278,Z 194.338,A -85,B 0,C 180,E1 -5834.174,E2 -5834.174} C_VEL
LIN {X 0,Y 504.301,Z 200.937,A -85,B 0,C 180,E1 -5834.336,E2 -5834.336} C_VEL
LIN {X 0,Y 505.389,Z 208.876,A -85,B 0,C 180,E1 -5834.486,E2 -5834.486} C_VEL
LIN {X 0,Y 504.86,Z 302.069,A -85,B 0,C 180,E1 -5835.848,E2 -5835.848} C_VEL
LIN {X 0,Y 504.588,Z 315.335,A -85,B 0,C 180,E1 -5836.2,E2 -5836.2} C_VEL
LIN {X 0,Y 504.234,Z 328.067,A -85,B 0,C 180,E1 -5836.704,E2 -5836.704} C_VEL
LIN {X 0,Y 503.952,Z 339.066,A -85,B 0,C 180,E1 -5837.291,E2 -5837.291} C_VEL
LIN {X 0,Y 503.643,Z 349.77,A -85,B 0,C 180,E1 -5838.019,E2 -5838.019} C_VEL
LIN {X 0,Y 503.284,Z 360.492,A -85,B 0,C 180,E1 -5838.929,E2 -5838.929} C_VEL
LIN {X 0,Y 502.9,Z 370.144,A -85,B 0,C 180,E1 -5839.939,E2 -5839.939} C_VEL
LIN {X 0,Y 502.649,Z 378.056,A -85,B 0,C 180,E1 -5840.949,E2 -5840.949} C_VEL
LIN {X 0,Y 502.412,Z 385.782,A -85,B 0,C 180,E1 -5842.16,E2 -5842.16} C_VEL
LIN {X 0,Y 502.237,Z 392.891,A -85,B 0,C 180,E1 -5843.572,E2 -5843.572} C_VEL
LIN {X 0,Y 502.18,Z 397.622,A -85,B 0,C 180,E1 -5844.78,E2 -5844.78} C_VEL
LIN {X 0,Y 502.139,Z 401.235,A -85,B 0,C 180,E1 -5845.986,E2 -5845.986} C_VEL
LIN {X 0,Y 502.121,Z 403.099,A -85,B 0,C 180,E1 -5846.79,E2 -5846.79} C_VEL
LIN {X 0,Y 502.066,Z 404.496,A -85,B 0,C 180,E1 -5847.592,E2 -5847.592} C_VEL
LIN {X 0,Y 502.036,Z 405.491,A -85,B 0,C 180,E1 -5848.395,E2 -5848.395} C_VEL
LIN {X 0,Y 501.981,Z 406.314,A -85,B 0,C 180,E1 -5849.999,E2 -5849.999} C_VEL
LIN {X 0,Y 502.036,Z 405.488,A -85,B 0,C 180,E1 -5851.604,E2 -5851.604} C_VEL
LIN {X 0,Y 502.066,Z 404.49,A -85,B 0,C 180,E1 -5852.406,E2 -5852.406} C_VEL
LIN {X 0,Y 502.12,Z 403.091,A -85,B 0,C 180,E1 -5853.209,E2 -5853.209} C_VEL
LIN {X 0,Y 502.102,Z 400.149,A -85,B 0,C 180,E1 -5854.414,E2 -5854.414} C_VEL
LIN {X 0,Y 502.228,Z 396.168,A -85,B 0,C 180,E1 -5855.621,E2 -5855.621} C_VEL
LIN {X 0,Y 502.332,Z 390.139,A -85,B 0,C 180,E1 -5857.011,E2 -5857.011} C_VEL
LIN {X 0,Y 502.471,Z 383.34,A -85,B 0,C 180,E1 -5858.242,E2 -5858.242} C_VEL
LIN {X 0,Y 502.734,Z 375.03,A -85,B 0,C 180,E1 -5859.453,E2 -5859.453} C_VEL
LIN {X 0,Y 502.996,Z 366.495,A -85,B 0,C 180,E1 -5860.464,E2 -5860.464} C_VEL
LIN {X 0,Y 503.398,Z 355.952,A -85,B 0,C 180,E1 -5861.474,E2 -5861.474} C_VEL
LIN {X 0,Y 503.733,Z 345.217,A -85,B 0,C 180,E1 -5862.304,E2 -5862.304} C_VEL
LIN {X 0,Y 504.094,Z 334.041,A -85,B 0,C 180,E1 -5862.991,E2 -5862.991} C_VEL
LIN {X 0,Y 504.413,Z 322.176,A -85,B 0,C 180,E1 -5863.546,E2 -5863.546} C_VEL
LIN {X 0,Y 504.695,Z 308.486,A -85,B 0,C 180,E1 -5864.001,E2 -5864.001} C_VEL
LIN {X 0,Y 504.901,Z 296.184,A -85,B 0,C 180,E1 -5864.252,E2 -5864.252} C_VEL
LIN {X 0,Y 505.325,Z 207.179,A -85,B 0,C 180,E1 -5865.543,E2 -5865.543} C_VEL
LIN {X 0,Y 503.285,Z 194.292,A -85,B 0,C 180,E1 -5865.824,E2 -5865.824} C_VEL
LIN {X 0,Y 503.726,Z 176.987,A -85,B 0,C 180,E1 -5868.716,E2 -5868.716} C_VEL
LIN {X 0,Y 504.234,Z 158.545,A -85,B 0,C 180,E1 -5871.89,E2 -5871.89} C_VEL
LIN {X 0,Y 504.152,Z 154.85,A -85,B 0,C 180,E1 -5872.54,E2 -5872.54} C_VEL
LIN {X 0,Y 502.829,Z 147.429,A -85,B 0,C 180,E1 -5873.965,E2 -5873.965} C_VEL
LIN {X 0,Y 502.78,Z 147.355,A -85,B 0,C 180,E1 -5876.57,E2 -5876.57} C_VEL
LIN {X 0,Y 502.748,Z 147.362,A -85,B 0,C 180,E1 -5879.291,E2 -5879.291} C_VEL
LIN {X 0,Y 502.768,Z 147.357,A -85,B 0,C 180,E1 -5882.084,E2 -5882.084} C_VEL
LIN {X 0,Y 502.777,Z 147.356,A -85,B 0,C 180,E1 -5884.966,E2 -5884.966} C_VEL
LIN {X 0,Y 502.747,Z 147.356,A -85,B 0,C 180,E1 -5888.479,E2 -5888.479} C_VEL
LIN {X 0,Y 502.754,Z 147.36,A -85,B 0,C 180,E1 -5891.071,E2 -5891.071} C_VEL
LIN {X 0,Y 502.769,Z 147.353,A -85,B 0,C 180,E1 -5894.528,E2 -5894.528} C_VEL
LIN {X 0,Y 502.757,Z 147.357,A -85,B 0,C 180,E1 -5897.856,E2 -5897.856} C_VEL
LIN {X 0,Y 502.772,Z 147.359,A -85,B 0,C 180,E1 -5901.021,E2 -5901.021} C_VEL
LIN {X 0,Y 502.758,Z 147.355,A -85,B 0,C 180,E1 -5904.169,E2 -5904.169} C_VEL
LIN {X 0,Y 502.788,Z 147.357,A -85,B 0,C 180,E1 -5906.998,E2 -5906.998} C_VEL
LIN {X 0,Y 502.778,Z 147.352,A -85,B 0,C 180,E1 -5910.069,E2 -5910.069} C_VEL
LIN {X 0,Y 502.764,Z 147.356,A -85,B 0,C 180,E1 -5912.529,E2 -5912.529} C_VEL
LIN {X 0,Y 502.758,Z 147.358,A -85,B 0,C 180,E1 -5915.313,E2 -5915.313} C_VEL
LIN {X 0,Y 502.766,Z 147.353,A -85,B 0,C 180,E1 -5917.825,E2 -5917.825} C_VEL
LIN {X 0,Y 502.798,Z 147.351,A -85,B 0,C 180,E1 -5920.399,E2 -5920.399} C_VEL
LIN {X 0,Y 502.792,Z 147.357,A -85,B 0,C 180,E1 -5922.93,E2 -5922.93} C_VEL
LIN {X 0,Y 502.81,Z 147.349,A -85,B 0,C 180,E1 -5925.428,E2 -5925.428} C_VEL
LIN {X 0,Y 502.859,Z 147.347,A -85,B 0,C 180,E1 -5928.716,E2 -5928.716} C_VEL
LIN {X 0,Y 502.864,Z 147.342,A -85,B 0,C 180,E1 -5931.966,E2 -5931.966} C_VEL
LIN {X 0,Y 502.902,Z 147.341,A -85,B 0,C 180,E1 -5934.386,E2 -5934.386} C_VEL
LIN {X 0,Y 502.997,Z 147.325,A -85,B 0,C 180,E1 -5937.597,E2 -5937.597} C_VEL
LIN {X 0,Y 502.995,Z 147.331,A -85,B 0,C 180,E1 -5940.8,E2 -5940.8} C_VEL
LIN {X 0,Y 502.996,Z 147.333,A -85,B 0,C 180,E1 -5942.402,E2 -5942.402} C_VEL
LIN {X 0,Y 502.903,Z 147.337,A -85,B 0,C 180,E1 -5945.614,E2 -5945.614} C_VEL
LIN {X 0,Y 502.856,Z 147.346,A -85,B 0,C 180,E1 -5948.034,E2 -5948.034} C_VEL
LIN {X 0,Y 502.821,Z 147.347,A -85,B 0,C 180,E1 -5951.284,E2 -5951.284} C_VEL
LIN {X 0,Y 502.819,Z 147.353,A -85,B 0,C 180,E1 -5954.571,E2 -5954.571} C_VEL
LIN {X 0,Y 502.785,Z 147.356,A -85,B 0,C 180,E1 -5957.909,E2 -5957.909} C_VEL
LIN {X 0,Y 502.815,Z 147.353,A -85,B 0,C 180,E1 -5960.536,E2 -5960.536} C_VEL
LIN {X 0,Y 502.772,Z 147.355,A -85,B 0,C 180,E1 -5963.041,E2 -5963.041} C_VEL
LIN {X 0,Y 502.761,Z 147.357,A -85,B 0,C 180,E1 -5965.679,E2 -5965.679} C_VEL
LIN {X 0,Y 502.755,Z 147.362,A -85,B 0,C 180,E1 -5968.377,E2 -5968.377} C_VEL
LIN {X 0,Y 502.778,Z 147.358,A -85,B 0,C 180,E1 -5971.144,E2 -5971.144} C_VEL
LIN {X 0,Y 502.866,Z 147.566,A -85,B 0,C 180,E1 -5972.315,E2 -5972.315} C_VEL
LIN {X 0,Y 503.853,Z 154.612,A -85,B 0,C 180,E1 -5973.683,E2 -5973.683} C_VEL
LIN {X 0,Y 503.472,Z 170.794,A -85,B 0,C 180,E1 -5976.637,E2 -5976.637} C_VEL
LIN {X 0,Y 503.294,Z 179.702,A -85,B 0,C 180,E1 -5978.218,E2 -5978.218} C_VEL
LIN {X 0,Y 505.383,Z 191.572,A -85,B 0,C 180,E1 -5978.494,E2 -5978.494} C_VEL
LIN {X 0,Y 504.832,Z 287.099,A -85,B 0,C 180,E1 -5979.899,E2 -5979.899} C_VEL
LIN {X 0,Y 504.615,Z 300.209,A -85,B 0,C 180,E1 -5980.251,E2 -5980.251} C_VEL
LIN {X 0,Y 504.355,Z 312.487,A -85,B 0,C 180,E1 -5980.739,E2 -5980.739} C_VEL
LIN {X 0,Y 504.077,Z 322.618,A -85,B 0,C 180,E1 -5981.273,E2 -5981.273} C_VEL
LIN {X 0,Y 503.254,Z 327.836,A -85,B 0,C 180,E1 -5981.575,E2 -5981.575} C_VEL
LIN {X 0,Y 500.155,Z 336.078,A -85,B 0,C 180,E1 -5982.098,E2 -5982.098} C_VEL
LIN {X 0,Y 497.056,Z 343.869,A -85,B 0,C 180,E1 -5982.703,E2 -5982.703} C_VEL
LIN {X 0,Y 496.239,Z 348.377,A -85,B 0,C 180,E1 -5983.132,E2 -5983.132} C_VEL
LIN {X 0,Y 495.831,Z 358.482,A -85,B 0,C 180,E1 -5984.294,E2 -5984.294} C_VEL
LIN {X 0,Y 495.554,Z 365.995,A -85,B 0,C 180,E1 -5985.358,E2 -5985.358} C_VEL
LIN {X 0,Y 495.393,Z 371.776,A -85,B 0,C 180,E1 -5986.345,E2 -5986.345} C_VEL
LIN {X 0,Y 495.239,Z 377.61,A -85,B 0,C 180,E1 -5987.555,E2 -5987.555} C_VEL
LIN {X 0,Y 495.127,Z 382.317,A -85,B 0,C 180,E1 -5988.789,E2 -5988.789} C_VEL
LIN {X 0,Y 494.984,Z 386.546,A -85,B 0,C 180,E1 -5990.29,E2 -5990.29} C_VEL
LIN {X 0,Y 494.92,Z 388.642,A -85,B 0,C 180,E1 -5991.353,E2 -5991.353} C_VEL
LIN {X 0,Y 494.834,Z 390.273,A -85,B 0,C 180,E1 -5992.688,E2 -5992.688} C_VEL
LIN {X 0,Y 494.869,Z 390.822,A -85,B 0,C 180,E1 -5994.046,E2 -5994.046} C_VEL
LIN {X 0,Y 494.866,Z 390.209,A -85,B 0,C 180,E1 -5995.457,E2 -5995.457} C_VEL
LIN {X 0,Y 494.935,Z 388.32,A -85,B 0,C 180,E1 -5996.907,E2 -5996.907} C_VEL
LIN {X 0,Y 495.062,Z 384.998,A -85,B 0,C 180,E1 -5998.404,E2 -5998.404} C_VEL
LIN {X 0,Y 495.124,Z 381.051,A -85,B 0,C 180,E1 -5999.655,E2 -5999.655} C_VEL
LIN {X 0,Y 495.304,Z 375.843,A -85,B 0,C 180,E1 -6000.925,E2 -6000.925} C_VEL
LIN {X 0,Y 495.479,Z 369.828,A -85,B 0,C 180,E1 -6002.092,E2 -6002.092} C_VEL
LIN {X 0,Y 495.687,Z 362.239,A -85,B 0,C 180,E1 -6003.281,E2 -6003.281} C_VEL
LIN {X 0,Y 496.058,Z 352.47,A -85,B 0,C 180,E1 -6004.512,E2 -6004.512} C_VEL
LIN {X 0,Y 496.465,Z 342.234,A -85,B 0,C 180,E1 -6005.544,E2 -6005.544} C_VEL
LIN {X 0,Y 496.872,Z 330.962,A -85,B 0,C 180,E1 -6006.449,E2 -6006.449} C_VEL
LIN {X 0,Y 497.208,Z 320.312,A -85,B 0,C 180,E1 -6007.131,E2 -6007.131} C_VEL
LIN {X 0,Y 497.548,Z 307.833,A -85,B 0,C 180,E1 -6007.746,E2 -6007.746} C_VEL
LIN {X 0,Y 497.831,Z 294.873,A -85,B 0,C 180,E1 -6008.196,E2 -6008.196} C_VEL
LIN {X 0,Y 498.039,Z 282.013,A -85,B 0,C 180,E1 -6008.477,E2 -6008.477} C_VEL
LIN {X 0,Y 498.534,Z 192.236,A -85,B 0,C 180,E1 -6009.796,E2 -6009.796} C_VEL
LIN {X 0,Y 496.388,Z 180.425,A -85,B 0,C 180,E1 -6010.056,E2 -6010.056} C_VEL
LIN {X 0,Y 496.337,Z 179.518,A -85,B 0,C 180,E1 -6010.134,E2 -6010.134} C_VEL
LIN {X 0,Y 496.76,Z 163.713,A -85,B 0,C 180,E1 -6013.142,E2 -6013.142} C_VEL
LIN {X 0,Y 496.989,Z 154.963,A -85,B 0,C 180,E1 -6014.835,E2 -6014.835} C_VEL
LIN {X 0,Y 495.861,Z 148.519,A -85,B 0,C 180,E1 -6016.163,E2 -6016.163} C_VEL
LIN {X 0,Y 495.795,Z 148.223,A -85,B 0,C 180,E1 -6016.475,E2 -6016.475} C_VEL
LIN {X 0,Y 495.775,Z 148.23,A -85,B 0,C 180,E1 -6019.382,E2 -6019.382} C_VEL
LIN {X 0,Y 495.87,Z 148.22,A -85,B 0,C 180,E1 -6021.853,E2 -6021.853} C_VEL
LIN {X 0,Y 495.892,Z 148.213,A -85,B 0,C 180,E1 -6024.307,E2 -6024.307} C_VEL
LIN {X 0,Y 495.99,Z 148.203,A -85,B 0,C 180,E1 -6027.565,E2 -6027.565} C_VEL
LIN {X 0,Y 495.995,Z 148.202,A -85,B 0,C 180,E1 -6030.001,E2 -6030.001} C_VEL
LIN {X 0,Y 495.99,Z 148.198,A -85,B 0,C 180,E1 -6032.437,E2 -6032.437} C_VEL
LIN {X 0,Y 495.886,Z 148.218,A -85,B 0,C 180,E1 -6035.694,E2 -6035.694} C_VEL
LIN {X 0,Y 495.835,Z 148.218,A -85,B 0,C 180,E1 -6038.149,E2 -6038.149} C_VEL
LIN {X 0,Y 495.85,Z 148.223,A -85,B 0,C 180,E1 -6041.446,E2 -6041.446} C_VEL
LIN {X 0,Y 495.788,Z 148.224,A -85,B 0,C 180,E1 -6044.784,E2 -6044.784} C_VEL
LIN {X 0,Y 495.763,Z 148.234,A -85,B 0,C 180,E1 -6047.32,E2 -6047.32} C_VEL
LIN {X 0,Y 495.77,Z 148.226,A -85,B 0,C 180,E1 -6049.891,E2 -6049.891} C_VEL
LIN {X 0,Y 495.758,Z 148.23,A -85,B 0,C 180,E1 -6052.861,E2 -6052.861} C_VEL
LIN {X 0,Y 495.779,Z 148.224,A -85,B 0,C 180,E1 -6056.069,E2 -6056.069} C_VEL
LIN {X 0,Y 495.768,Z 148.229,A -85,B 0,C 180,E1 -6058.815,E2 -6058.815} C_VEL
LIN {X 0,Y 495.753,Z 148.228,A -85,B 0,C 180,E1 -6061.726,E2 -6061.726} C_VEL
LIN {X 0,Y 495.761,Z 148.23,A -85,B 0,C 180,E1 -6064.693,E2 -6064.693} C_VEL
LIN {X 0,Y 495.727,Z 148.231,A -85,B 0,C 180,E1 -6067.562,E2 -6067.562} C_VEL
LIN {X 0,Y 495.764,Z 148.232,A -85,B 0,C 180,E1 -6070.7,E2 -6070.7} C_VEL
LIN {X 0,Y 495.727,Z 148.231,A -85,B 0,C 180,E1 -6074.002,E2 -6074.002} C_VEL
LIN {X 0,Y 495.716,Z 148.235,A -85,B 0,C 180,E1 -6077.116,E2 -6077.116} C_VEL
LIN {X 0,Y 495.757,Z 148.227,A -85,B 0,C 180,E1 -6079.954,E2 -6079.954} C_VEL
LIN {X 0,Y 495.717,Z 148.24,A -85,B 0,C 180,E1 -6082.555,E2 -6082.555} C_VEL
LIN {X 0,Y 495.776,Z 148.224,A -85,B 0,C 180,E1 -6085.457,E2 -6085.457} C_VEL
LIN {X 0,Y 495.754,Z 148.234,A -85,B 0,C 180,E1 -6088.364,E2 -6088.364} C_VEL
LIN {X 0,Y 495.753,Z 148.227,A -85,B 0,C 180,E1 -6091.515,E2 -6091.515} C_VEL
LIN {X 0,Y 495.756,Z 148.23,A -85,B 0,C 180,E1 -6093.931,E2 -6093.931} C_VEL
LIN {X 0,Y 495.757,Z 148.227,A -85,B 0,C 180,E1 -6097.14,E2 -6097.14} C_VEL
LIN {X 0,Y 495.766,Z 148.232,A -85,B 0,C 180,E1 -6100.11,E2 -6100.11} C_VEL
LIN {X 0,Y 495.753,Z 148.229,A -85,B 0,C 180,E1 -6102.681,E2 -6102.681} C_VEL
LIN {X 0,Y 495.781,Z 148.224,A -85,B 0,C 180,E1 -6105.217,E2 -6105.217} C_VEL
LIN {X 0,Y 495.85,Z 148.217,A -85,B 0,C 180,E1 -6108.555,E2 -6108.555} C_VEL
LIN {X 0,Y 495.814,Z 148.226,A -85,B 0,C 180,E1 -6111.851,E2 -6111.851} C_VEL
LIN {X 0,Y 495.854,Z 148.218,A -85,B 0,C 180,E1 -6114.306,E2 -6114.306} C_VEL
LIN {X 0,Y 495.975,Z 148.204,A -85,B 0,C 180,E1 -6117.564,E2 -6117.564} C_VEL
LIN {X 0,Y 495.97,Z 148.205,A -85,B 0,C 180,E1 -6120,E2 -6120} C_VEL
LIN {X 0,Y 495.981,Z 148.199,A -85,B 0,C 180,E1 -6122.437,E2 -6122.437} C_VEL
LIN {X 0,Y 495.845,Z 148.224,A -85,B 0,C 180,E1 -6125.694,E2 -6125.694} C_VEL
LIN {X 0,Y 495.812,Z 148.221,A -85,B 0,C 180,E1 -6128.149,E2 -6128.149} C_VEL
LIN {X 0,Y 495.849,Z 148.222,A -85,B 0,C 180,E1 -6131.446,E2 -6131.446} C_VEL
LIN {X 0,Y 495.774,Z 148.225,A -85,B 0,C 180,E1 -6134.784,E2 -6134.784} C_VEL
LIN {X 0,Y 495.773,Z 148.225,A -85,B 0,C 180,E1 -6138.235,E2 -6138.235} C_VEL
LIN {X 0,Y 495.775,Z 148.226,A -85,B 0,C 180,E1 -6140.757,E2 -6140.757} C_VEL
LIN {X 0,Y 495.735,Z 148.236,A -85,B 0,C 180,E1 -6143.388,E2 -6143.388} C_VEL
LIN {X 0,Y 495.707,Z 148.233,A -85,B 0,C 180,E1 -6146.073,E2 -6146.073} C_VEL
LIN {X 0,Y 495.696,Z 148.238,A -85,B 0,C 180,E1 -6148.82,E2 -6148.82} C_VEL
LIN {X 0,Y 495.731,Z 148.231,A -85,B 0,C 180,E1 -6151.72,E2 -6151.72} C_VEL
LIN {X 0,Y 495.753,Z 148.231,A -85,B 0,C 180,E1 -6154.691,E2 -6154.691} C_VEL
LIN {X 0,Y 495.7,Z 148.235,A -85,B 0,C 180,E1 -6157.565,E2 -6157.565} C_VEL
LIN {X 0,Y 495.71,Z 148.232,A -85,B 0,C 180,E1 -6160.04,E2 -6160.04} C_VEL
LIN {X 0,Y 495.691,Z 148.243,A -85,B 0,C 180,E1 -6162.887,E2 -6162.887} C_VEL
LIN {X 0,Y 495.714,Z 148.232,A -85,B 0,C 180,E1 -6165.997,E2 -6165.997} C_VEL
LIN {X 0,Y 495.71,Z 148.234,A -85,B 0,C 180,E1 -6169.294,E2 -6169.294} C_VEL
LIN {X 0,Y 495.707,Z 148.233,A -85,B 0,C 180,E1 -6171.404,E2 -6171.404} C_VEL
LIN {X 0,Y 495.69,Z 148.242,A -85,B 0,C 180,E1 -6174.457,E2 -6174.457} C_VEL
LIN {X 0,Y 495.724,Z 148.231,A -85,B 0,C 180,E1 -6177.402,E2 -6177.402} C_VEL
LIN {X 0,Y 495.698,Z 148.242,A -85,B 0,C 180,E1 -6180.249,E2 -6180.249} C_VEL
LIN {X 0,Y 495.724,Z 148.232,A -85,B 0,C 180,E1 -6183.275,E2 -6183.275} C_VEL
LIN {X 0,Y 495.816,Z 148.457,A -85,B 0,C 180,E1 -6185.811,E2 -6185.811} C_VEL
LIN {X 0,Y 497.406,Z 157.7,A -85,B 0,C 180,E1 -6187.573,E2 -6187.573} C_VEL
LIN {X 0,Y 496.96,Z 171.086,A -85,B 0,C 180,E1 -6189.943,E2 -6189.943} C_VEL
LIN {X 0,Y 496.469,Z 186.885,A -85,B 0,C 180,E1 -6192.705,E2 -6192.705} C_VEL
LIN {X 0,Y 496.293,Z 194.298,A -85,B 0,C 180,E1 -6193.953,E2 -6193.953} C_VEL
LIN {X 0,Y 498.069,Z 205.355,A -85,B 0,C 180,E1 -6194.206,E2 -6194.206} C_VEL
LIN {X 0,Y 498.507,Z 209.998,A -85,B 0,C 180,E1 -6194.289,E2 -6194.289} C_VEL
LIN {X 0,Y 497.994,Z 301.768,A -85,B 0,C 180,E1 -6195.649,E2 -6195.649} C_VEL
LIN {X 0,Y 497.678,Z 315.098,A -85,B 0,C 180,E1 -6196.005,E2 -6196.005} C_VEL
LIN {X 0,Y 497.319,Z 327.862,A -85,B 0,C 180,E1 -6196.515,E2 -6196.515} C_VEL
LIN {X 0,Y 497.01,Z 338.895,A -85,B 0,C 180,E1 -6197.111,E2 -6197.111} C_VEL
LIN {X 0,Y 496.671,Z 349.606,A -85,B 0,C 180,E1 -6197.849,E2 -6197.849} C_VEL
LIN {X 0,Y 496.294,Z 360.339,A -85,B 0,C 180,E1 -6198.771,E2 -6198.771} C_VEL
LIN {X 0,Y 495.862,Z 370,A -85,B 0,C 180,E1 -6199.795,E2 -6199.795} C_VEL
LIN {X 0,Y 495.611,Z 377.921,A -85,B 0,C 180,E1 -6200.82,E2 -6200.82} C_VEL
LIN {X 0,Y 495.355,Z 385.656,A -85,B 0,C 180,E1 -6202.048,E2 -6202.048} C_VEL
LIN {X 0,Y 495.135,Z 392.77,A -85,B 0,C 180,E1 -6203.479,E2 -6203.479} C_VEL
LIN {X 0,Y 495.114,Z 397.506,A -85,B 0,C 180,E1 -6204.705,E2 -6204.705} C_VEL
LIN {X 0,Y 495.033,Z 401.121,A -85,B 0,C 180,E1 -6205.929,E2 -6205.929} C_VEL
LIN {X 0,Y 495.042,Z 402.987,A -85,B 0,C 180,E1 -6206.744,E2 -6206.744} C_VEL
LIN {X 0,Y 494.961,Z 405.381,A -85,B 0,C 180,E1 -6208.372,E2 -6208.372} C_VEL
LIN {X 0,Y 494.899,Z 406.204,A -85,B 0,C 180,E1 -6209.999,E2 -6209.999} C_VEL
LIN {X 0,Y 494.961,Z 405.376,A -85,B 0,C 180,E1 -6211.626,E2 -6211.626} C_VEL
LIN {X 0,Y 495.042,Z 402.978,A -85,B 0,C 180,E1 -6213.255,E2 -6213.255} C_VEL
LIN {X 0,Y 495.007,Z 400.033,A -85,B 0,C 180,E1 -6214.478,E2 -6214.478} C_VEL
LIN {X 0,Y 495.145,Z 396.049,A -85,B 0,C 180,E1 -6215.701,E2 -6215.701} C_VEL
LIN {X 0,Y 495.256,Z 389.915,A -85,B 0,C 180,E1 -6217.132,E2 -6217.132} C_VEL
LIN {X 0,Y 495.421,Z 383.213,A -85,B 0,C 180,E1 -6218.36,E2 -6218.36} C_VEL
LIN {X 0,Y 495.715,Z 374.898,A -85,B 0,C 180,E1 -6219.588,E2 -6219.588} C_VEL
LIN {X 0,Y 495.991,Z 366.356,A -85,B 0,C 180,E1 -6220.614,E2 -6220.614} C_VEL
LIN {X 0,Y 496.42,Z 355.804,A -85,B 0,C 180,E1 -6221.638,E2 -6221.638} C_VEL
LIN {X 0,Y 496.79,Z 344.187,A -85,B 0,C 180,E1 -6222.543,E2 -6222.543} C_VEL
LIN {X 0,Y 497.183,Z 331.907,A -85,B 0,C 180,E1 -6223.279,E2 -6223.279} C_VEL
LIN {X 0,Y 497.567,Z 319.405,A -85,B 0,C 180,E1 -6223.84,E2 -6223.84} C_VEL
LIN {X 0,Y 497.849,Z 306.36,A -85,B 0,C 180,E1 -6224.249,E2 -6224.249} C_VEL
LIN {X 0,Y 498.038,Z 290.68,A -85,B 0,C 180,E1 -6224.531,E2 -6224.531} C_VEL
LIN {X 0,Y 498.412,Z 207.31,A -85,B 0,C 180,E1 -6225.765,E2 -6225.765} C_VEL
LIN {X 0,Y 496.319,Z 194.347,A -85,B 0,C 180,E1 -6226.043,E2 -6226.043} C_VEL
LIN {X 0,Y 496.378,Z 190.415,A -85,B 0,C 180,E1 -6226.66,E2 -6226.66} C_VEL
LIN {X 0,Y 496.819,Z 174.43,A -85,B 0,C 180,E1 -6229.415,E2 -6229.415} C_VEL
LIN {X 0,Y 497.352,Z 158.436,A -85,B 0,C 180,E1 -6232.209,E2 -6232.209} C_VEL
LIN {X 0,Y 496.3,Z 151.035,A -85,B 0,C 180,E1 -6233.579,E2 -6233.579} C_VEL
LIN {X 0,Y 495.795,Z 148.283,A -85,B 0,C 180,E1 -6234.16,E2 -6234.16} C_VEL
LIN {X 0,Y 495.725,Z 148.235,A -85,B 0,C 180,E1 -6236.978,E2 -6236.978} C_VEL
LIN {X 0,Y 495.693,Z 148.239,A -85,B 0,C 180,E1 -6240.132,E2 -6240.132} C_VEL
LIN {X 0,Y 495.746,Z 148.233,A -85,B 0,C 180,E1 -6243.235,E2 -6243.235} C_VEL
LIN {X 0,Y 495.68,Z 148.239,A -85,B 0,C 180,E1 -6246.082,E2 -6246.082} C_VEL
LIN {X 0,Y 495.725,Z 148.232,A -85,B 0,C 180,E1 -6248.762,E2 -6248.762} C_VEL
LIN {X 0,Y 495.716,Z 148.236,A -85,B 0,C 180,E1 -6251.783,E2 -6251.783} C_VEL
LIN {X 0,Y 495.723,Z 148.237,A -85,B 0,C 180,E1 -6255.14,E2 -6255.14} C_VEL
LIN {X 0,Y 495.714,Z 148.233,A -85,B 0,C 180,E1 -6258.214,E2 -6258.214} C_VEL
LIN {X 0,Y 495.73,Z 148.237,A -85,B 0,C 180,E1 -6261.234,E2 -6261.234} C_VEL
LIN {X 0,Y 495.731,Z 148.231,A -85,B 0,C 180,E1 -6264.461,E2 -6264.461} C_VEL
LIN {X 0,Y 495.729,Z 148.235,A -85,B 0,C 180,E1 -6267.402,E2 -6267.402} C_VEL
LIN {X 0,Y 495.727,Z 148.23,A -85,B 0,C 180,E1 -6270.251,E2 -6270.251} C_VEL
LIN {X 0,Y 495.727,Z 148.235,A -85,B 0,C 180,E1 -6273.269,E2 -6273.269} C_VEL
LIN {X 0,Y 495.725,Z 148.234,A -85,B 0,C 180,E1 -6276.611,E2 -6276.611} C_VEL
LIN {X 0,Y 495.767,Z 148.227,A -85,B 0,C 180,E1 -6279.323,E2 -6279.323} C_VEL
LIN {X 0,Y 495.766,Z 148.225,A -85,B 0,C 180,E1 -6281.828,E2 -6281.828} C_VEL
LIN {X 0,Y 495.81,Z 148.224,A -85,B 0,C 180,E1 -6284.548,E2 -6284.548} C_VEL
LIN {X 0,Y 495.815,Z 148.219,A -85,B 0,C 180,E1 -6287.965,E2 -6287.965} C_VEL
LIN {X 0,Y 495.814,Z 148.224,A -85,B 0,C 180,E1 -6291.029,E2 -6291.029} C_VEL
LIN {X 0,Y 495.833,Z 148.217,A -85,B 0,C 180,E1 -6293.489,E2 -6293.489} C_VEL
LIN {X 0,Y 495.796,Z 148.227,A -85,B 0,C 180,E1 -6296.749,E2 -6296.749} C_VEL
LIN {X 0,Y 495.856,Z 148.22,A -85,B 0,C 180,E1 -6298.375,E2 -6298.375} C_VEL
LIN {X 0,Y 495.946,Z 148.209,A -85,B 0,C 180,E1 -6300.812,E2 -6300.812} C_VEL
LIN {X 0,Y 495.964,Z 148.209,A -85,B 0,C 180,E1 -6302.436,E2 -6302.436} C_VEL
LIN {X 0,Y 495.86,Z 148.215,A -85,B 0,C 180,E1 -6305.694,E2 -6305.694} C_VEL
LIN {X 0,Y 495.813,Z 148.225,A -85,B 0,C 180,E1 -6308.149,E2 -6308.149} C_VEL
LIN {X 0,Y 495.806,Z 148.221,A -85,B 0,C 180,E1 -6311.446,E2 -6311.446} C_VEL
LIN {X 0,Y 495.767,Z 148.229,A -85,B 0,C 180,E1 -6314.783,E2 -6314.783} C_VEL
LIN {X 0,Y 495.764,Z 148.233,A -85,B 0,C 180,E1 -6318.172,E2 -6318.172} C_VEL
LIN {X 0,Y 495.76,Z 148.23,A -85,B 0,C 180,E1 -6320.757,E2 -6320.757} C_VEL
LIN {X 0,Y 495.724,Z 148.233,A -85,B 0,C 180,E1 -6323.388,E2 -6323.388} C_VEL
LIN {X 0,Y 495.723,Z 148.234,A -85,B 0,C 180,E1 -6326.73,E2 -6326.73} C_VEL
LIN {X 0,Y 495.742,Z 148.235,A -85,B 0,C 180,E1 -6329.747,E2 -6329.747} C_VEL
LIN {X 0,Y 495.8,Z 148.356,A -85,B 0,C 180,E1 -6332.118,E2 -6332.118} C_VEL
LIN {X 0,Y 496.872,Z 155.15,A -85,B 0,C 180,E1 -6333.479,E2 -6333.479} C_VEL
LIN {X 0,Y 496.516,Z 171.361,A -85,B 0,C 180,E1 -6336.476,E2 -6336.476} C_VEL
LIN {X 0,Y 496.352,Z 179.806,A -85,B 0,C 180,E1 -6337.986,E2 -6337.986} C_VEL
LIN {X 0,Y 498.613,Z 193.215,A -85,B 0,C 180,E1 -6338.297,E2 -6338.297} C_VEL
LIN {X 0,Y 497.952,Z 287.469,A -85,B 0,C 180,E1 -6339.707,E2 -6339.707} C_VEL
LIN {X 0,Y 497.728,Z 300.794,A -85,B 0,C 180,E1 -6340.075,E2 -6340.075} C_VEL
LIN {X 0,Y 497.428,Z 313.653,A -85,B 0,C 180,E1 -6340.602,E2 -6340.602} C_VEL
LIN {X 0,Y 497.016,Z 325.619,A -85,B 0,C 180,E1 -6341.272,E2 -6341.272} C_VEL
LIN {X 0,Y 496.682,Z 336.161,A -85,B 0,C 180,E1 -6342.026,E2 -6342.026} C_VEL
LIN {X 0,Y 496.291,Z 346.978,A -85,B 0,C 180,E1 -6342.988,E2 -6342.988} C_VEL
LIN {X 0,Y 496.239,Z 348.377,A -85,B 0,C 180,E1 -6343.132,E2 -6343.132} C_VEL
LIN {X 0,Y 495.423,Z 352.758,A -85,B 0,C 180,E1 -6343.587,E2 -6343.587} C_VEL
LIN {X 0,Y 492.313,Z 359.529,A -85,B 0,C 180,E1 -6344.352,E2 -6344.352} C_VEL
LIN {X 0,Y 489.222,Z 365.694,A -85,B 0,C 180,E1 -6345.182,E2 -6345.182} C_VEL
LIN {X 0,Y 488.437,Z 369.123,A -85,B 0,C 180,E1 -6345.734,E2 -6345.734} C_VEL
LIN {X 0,Y 488.257,Z 374.756,A -85,B 0,C 180,E1 -6346.805,E2 -6346.805} C_VEL
LIN {X 0,Y 488.096,Z 379.767,A -85,B 0,C 180,E1 -6347.971,E2 -6347.971} C_VEL
LIN {X 0,Y 487.99,Z 385.088,A -85,B 0,C 180,E1 -6349.604,E2 -6349.604} C_VEL
LIN {X 0,Y 487.829,Z 388.333,A -85,B 0,C 180,E1 -6351.074,E2 -6351.074} C_VEL
LIN {X 0,Y 487.755,Z 390.455,A -85,B 0,C 180,E1 -6352.761,E2 -6352.761} C_VEL
LIN {X 0,Y 487.765,Z 390.89,A -85,B 0,C 180,E1 -6353.791,E2 -6353.791} C_VEL
LIN {X 0,Y 487.759,Z 390.512,A -85,B 0,C 180,E1 -6355.214,E2 -6355.214} C_VEL
LIN {X 0,Y 487.827,Z 388.672,A -85,B 0,C 180,E1 -6356.809,E2 -6356.809} C_VEL
LIN {X 0,Y 487.943,Z 385.819,A -85,B 0,C 180,E1 -6358.189,E2 -6358.189} C_VEL
LIN {X 0,Y 488.039,Z 381.031,A -85,B 0,C 180,E1 -6359.771,E2 -6359.771} C_VEL
LIN {X 0,Y 488.248,Z 375.65,A -85,B 0,C 180,E1 -6361.088,E2 -6361.088} C_VEL
LIN {X 0,Y 488.452,Z 369.061,A -85,B 0,C 180,E1 -6362.354,E2 -6362.354} C_VEL
LIN {X 0,Y 488.704,Z 361.519,A -85,B 0,C 180,E1 -6363.526,E2 -6363.526} C_VEL
LIN {X 0,Y 489.088,Z 352.279,A -85,B 0,C 180,E1 -6364.693,E2 -6364.693} C_VEL
LIN {X 0,Y 489.496,Z 342.01,A -85,B 0,C 180,E1 -6365.734,E2 -6365.734} C_VEL
LIN {X 0,Y 489.916,Z 330.711,A -85,B 0,C 180,E1 -6366.649,E2 -6366.649} C_VEL
LIN {X 0,Y 490.338,Z 318.907,A -85,B 0,C 180,E1 -6367.401,E2 -6367.401} C_VEL
LIN {X 0,Y 490.65,Z 307.097,A -85,B 0,C 180,E1 -6367.97,E2 -6367.97} C_VEL
LIN {X 0,Y 490.952,Z 293.508,A -85,B 0,C 180,E1 -6368.434,E2 -6368.434} C_VEL
LIN {X 0,Y 491.157,Z 280.369,A -85,B 0,C 180,E1 -6368.706,E2 -6368.706} C_VEL
LIN {X 0,Y 491.601,Z 192.594,A -85,B 0,C 180,E1 -6370.017,E2 -6370.017} C_VEL
LIN {X 0,Y 489.37,Z 180.163,A -85,B 0,C 180,E1 -6370.304,E2 -6370.304} C_VEL
LIN {X 0,Y 489.437,Z 176.705,A -85,B 0,C 180,E1 -6370.909,E2 -6370.909} C_VEL
LIN {X 0,Y 490.032,Z 159.836,A -85,B 0,C 180,E1 -6374.188,E2 -6374.188} C_VEL
LIN {X 0,Y 489.776,Z 154.565,A -85,B 0,C 180,E1 -6375.245,E2 -6375.245} C_VEL
LIN {X 0,Y 488.787,Z 149.233,A -85,B 0,C 180,E1 -6376.383,E2 -6376.383} C_VEL
LIN {X 0,Y 488.737,Z 149.106,A -85,B 0,C 180,E1 -6379.227,E2 -6379.227} C_VEL
LIN {X 0,Y 488.859,Z 149.087,A -85,B 0,C 180,E1 -6382.567,E2 -6382.567} C_VEL
LIN {X 0,Y 488.807,Z 149.093,A -85,B 0,C 180,E1 -6385.052,E2 -6385.052} C_VEL
LIN {X 0,Y 488.957,Z 149.078,A -85,B 0,C 180,E1 -6387.53,E2 -6387.53} C_VEL
LIN {X 0,Y 488.966,Z 149.077,A -85,B 0,C 180,E1 -6390.001,E2 -6390.001} C_VEL
LIN {X 0,Y 488.958,Z 149.074,A -85,B 0,C 180,E1 -6392.472,E2 -6392.472} C_VEL
LIN {X 0,Y 488.845,Z 149.094,A -85,B 0,C 180,E1 -6395.777,E2 -6395.777} C_VEL
LIN {X 0,Y 488.784,Z 149.096,A -85,B 0,C 180,E1 -6398.268,E2 -6398.268} C_VEL
LIN {X 0,Y 488.804,Z 149.1,A -85,B 0,C 180,E1 -6401.613,E2 -6401.613} C_VEL
LIN {X 0,Y 488.76,Z 149.101,A -85,B 0,C 180,E1 -6405.001,E2 -6405.001} C_VEL
LIN {X 0,Y 488.746,Z 149.1,A -85,B 0,C 180,E1 -6408.443,E2 -6408.443} C_VEL
LIN {X 0,Y 488.706,Z 149.11,A -85,B 0,C 180,E1 -6411.071,E2 -6411.071} C_VEL
LIN {X 0,Y 488.675,Z 149.111,A -85,B 0,C 180,E1 -6413.747,E2 -6413.747} C_VEL
LIN {X 0,Y 488.79,Z 149.1,A -85,B 0,C 180,E1 -6416.944,E2 -6416.944} C_VEL
LIN {X 0,Y 488.707,Z 149.105,A -85,B 0,C 180,E1 -6420.363,E2 -6420.363} C_VEL
LIN {X 0,Y 488.728,Z 149.105,A -85,B 0,C 180,E1 -6423.484,E2 -6423.484} C_VEL
LIN {X 0,Y 488.681,Z 149.109,A -85,B 0,C 180,E1 -6426.355,E2 -6426.355} C_VEL
LIN {X 0,Y 488.696,Z 149.11,A -85,B 0,C 180,E1 -6429.255,E2 -6429.255} C_VEL
LIN {X 0,Y 488.705,Z 149.105,A -85,B 0,C 180,E1 -6431.6,E2 -6431.6} C_VEL
LIN {X 0,Y 488.7,Z 149.114,A -85,B 0,C 180,E1 -6434.803,E2 -6434.803} C_VEL
LIN {X 0,Y 488.687,Z 149.108,A -85,B 0,C 180,E1 -6437.475,E2 -6437.475} C_VEL
LIN {X 0,Y 488.699,Z 149.113,A -85,B 0,C 180,E1 -6440.746,E2 -6440.746} C_VEL
LIN {X 0,Y 488.668,Z 149.11,A -85,B 0,C 180,E1 -6443.868,E2 -6443.868} C_VEL
LIN {X 0,Y 488.737,Z 149.104,A -85,B 0,C 180,E1 -6446.878,E2 -6446.878} C_VEL
LIN {X 0,Y 488.722,Z 149.104,A -85,B 0,C 180,E1 -6449.781,E2 -6449.781} C_VEL
LIN {X 0,Y 488.723,Z 149.104,A -85,B 0,C 180,E1 -6453.073,E2 -6453.073} C_VEL
LIN {X 0,Y 488.674,Z 149.117,A -85,B 0,C 180,E1 -6456.254,E2 -6456.254} C_VEL
LIN {X 0,Y 488.746,Z 149.1,A -85,B 0,C 180,E1 -6459.176,E2 -6459.176} C_VEL
LIN {X 0,Y 488.747,Z 149.102,A -85,B 0,C 180,E1 -6461.633,E2 -6461.633} C_VEL
LIN {X 0,Y 488.756,Z 149.099,A -85,B 0,C 180,E1 -6465,E2 -6465} C_VEL
LIN {X 0,Y 488.804,Z 149.096,A -85,B 0,C 180,E1 -6468.388,E2 -6468.388} C_VEL
LIN {X 0,Y 488.762,Z 149.103,A -85,B 0,C 180,E1 -6471.733,E2 -6471.733} C_VEL
LIN {X 0,Y 488.814,Z 149.096,A -85,B 0,C 180,E1 -6474.224,E2 -6474.224} C_VEL
LIN {X 0,Y 488.941,Z 149.08,A -85,B 0,C 180,E1 -6477.529,E2 -6477.529} C_VEL
LIN {X 0,Y 488.939,Z 149.081,A -85,B 0,C 180,E1 -6480,E2 -6480} C_VEL
LIN {X 0,Y 488.948,Z 149.075,A -85,B 0,C 180,E1 -6482.472,E2 -6482.472} C_VEL
LIN {X 0,Y 488.804,Z 149.1,A -85,B 0,C 180,E1 -6485.777,E2 -6485.777} C_VEL
LIN {X 0,Y 488.759,Z 149.099,A -85,B 0,C 180,E1 -6488.268,E2 -6488.268} C_VEL
LIN {X 0,Y 488.804,Z 149.1,A -85,B 0,C 180,E1 -6491.613,E2 -6491.613} C_VEL
LIN {X 0,Y 488.752,Z 149.102,A -85,B 0,C 180,E1 -6495.001,E2 -6495.001} C_VEL
LIN {X 0,Y 488.745,Z 149.1,A -85,B 0,C 180,E1 -6498.443,E2 -6498.443} C_VEL
LIN {X 0,Y 488.706,Z 149.11,A -85,B 0,C 180,E1 -6501.071,E2 -6501.071} C_VEL
LIN {X 0,Y 488.663,Z 149.113,A -85,B 0,C 180,E1 -6503.747,E2 -6503.747} C_VEL
LIN {X 0,Y 488.669,Z 149.11,A -85,B 0,C 180,E1 -6506.477,E2 -6506.477} C_VEL
LIN {X 0,Y 488.66,Z 149.117,A -85,B 0,C 180,E1 -6509.275,E2 -6509.275} C_VEL
LIN {X 0,Y 488.679,Z 149.108,A -85,B 0,C 180,E1 -6512.149,E2 -6512.149} C_VEL
LIN {X 0,Y 488.705,Z 149.112,A -85,B 0,C 180,E1 -6515.116,E2 -6515.116} C_VEL
LIN {X 0,Y 488.654,Z 149.112,A -85,B 0,C 180,E1 -6518.203,E2 -6518.203} C_VEL
LIN {X 0,Y 488.644,Z 149.114,A -85,B 0,C 180,E1 -6521.423,E2 -6521.423} C_VEL
LIN {X 0,Y 488.697,Z 149.115,A -85,B 0,C 180,E1 -6524.804,E2 -6524.804} C_VEL
LIN {X 0,Y 488.65,Z 149.113,A -85,B 0,C 180,E1 -6527.47,E2 -6527.47} C_VEL
LIN {X 0,Y 488.667,Z 149.118,A -85,B 0,C 180,E1 -6530.742,E2 -6530.742} C_VEL
LIN {X 0,Y 488.608,Z 149.118,A -85,B 0,C 180,E1 -6533.862,E2 -6533.862} C_VEL
LIN {X 0,Y 488.675,Z 149.113,A -85,B 0,C 180,E1 -6536.872,E2 -6536.872} C_VEL
LIN {X 0,Y 488.666,Z 149.113,A -85,B 0,C 180,E1 -6539.776,E2 -6539.776} C_VEL
LIN {X 0,Y 488.678,Z 149.116,A -85,B 0,C 180,E1 -6542.599,E2 -6542.599} C_VEL
LIN {X 0,Y 488.716,Z 149.21,A -85,B 0,C 180,E1 -6545.578,E2 -6545.578} C_VEL
LIN {X 0,Y 490.444,Z 158.799,A -85,B 0,C 180,E1 -6547.46,E2 -6547.46} C_VEL
LIN {X 0,Y 490.023,Z 170.966,A -85,B 0,C 180,E1 -6549.647,E2 -6549.647} C_VEL
LIN {X 0,Y 489.515,Z 186.763,A -85,B 0,C 180,E1 -6552.452,E2 -6552.452} C_VEL
LIN {X 0,Y 489.314,Z 194.096,A -85,B 0,C 180,E1 -6553.713,E2 -6553.713} C_VEL
LIN {X 0,Y 490.074,Z 199.084,A -85,B 0,C 180,E1 -6553.853,E2 -6553.853} C_VEL
LIN {X 0,Y 491.672,Z 209.636,A -85,B 0,C 180,E1 -6554.065,E2 -6554.065} C_VEL
LIN {X 0,Y 491.081,Z 302.558,A -85,B 0,C 180,E1 -6555.469,E2 -6555.469} C_VEL
LIN {X 0,Y 490.768,Z 315.585,A -85,B 0,C 180,E1 -6555.83,E2 -6555.83} C_VEL
LIN {X 0,Y 490.405,Z 327.632,A -85,B 0,C 180,E1 -6556.322,E2 -6556.322} C_VEL
LIN {X 0,Y 490.048,Z 339.307,A -85,B 0,C 180,E1 -6556.964,E2 -6556.964} C_VEL
LIN {X 0,Y 489.667,Z 350.731,A -85,B 0,C 180,E1 -6557.777,E2 -6557.777} C_VEL
LIN {X 0,Y 489.268,Z 361.256,A -85,B 0,C 180,E1 -6558.713,E2 -6558.713} C_VEL
LIN {X 0,Y 488.853,Z 369.856,A -85,B 0,C 180,E1 -6559.647,E2 -6559.647} C_VEL
LIN {X 0,Y 488.563,Z 377.783,A -85,B 0,C 180,E1 -6560.686,E2 -6560.686} C_VEL
LIN {X 0,Y 488.309,Z 385.528,A -85,B 0,C 180,E1 -6561.932,E2 -6561.932} C_VEL
LIN {X 0,Y 488.067,Z 392.647,A -85,B 0,C 180,E1 -6563.384,E2 -6563.384} C_VEL
LIN {X 0,Y 488.047,Z 397.387,A -85,B 0,C 180,E1 -6564.628,E2 -6564.628} C_VEL
LIN {X 0,Y 487.928,Z 401.005,A -85,B 0,C 180,E1 -6565.869,E2 -6565.869} C_VEL
LIN {X 0,Y 487.965,Z 402.874,A -85,B 0,C 180,E1 -6566.697,E2 -6566.697} C_VEL
LIN {X 0,Y 487.889,Z 405.27,A -85,B 0,C 180,E1 -6568.348,E2 -6568.348} C_VEL
LIN {X 0,Y 487.82,Z 406.094,A -85,B 0,C 180,E1 -6569.999,E2 -6569.999} C_VEL
LIN {X 0,Y 487.889,Z 405.266,A -85,B 0,C 180,E1 -6571.65,E2 -6571.65} C_VEL
LIN {X 0,Y 487.964,Z 402.865,A -85,B 0,C 180,E1 -6573.302,E2 -6573.302} C_VEL
LIN {X 0,Y 487.92,Z 399.918,A -85,B 0,C 180,E1 -6574.543,E2 -6574.543} C_VEL
LIN {X 0,Y 488.062,Z 395.931,A -85,B 0,C 180,E1 -6575.784,E2 -6575.784} C_VEL
LIN {X 0,Y 488.182,Z 389.793,A -85,B 0,C 180,E1 -6577.236,E2 -6577.236} C_VEL
LIN {X 0,Y 488.359,Z 383.089,A -85,B 0,C 180,E1 -6578.482,E2 -6578.482} C_VEL
LIN {X 0,Y 488.698,Z 374.772,A -85,B 0,C 180,E1 -6579.727,E2 -6579.727} C_VEL
LIN {X 0,Y 488.999,Z 366.228,A -85,B 0,C 180,E1 -6580.767,E2 -6580.767} C_VEL
LIN {X 0,Y 489.447,Z 355.676,A -85,B 0,C 180,E1 -6581.806,E2 -6581.806} C_VEL
LIN {X 0,Y 489.833,Z 344.111,A -85,B 0,C 180,E1 -6582.72,E2 -6582.72} C_VEL
LIN {X 0,Y 490.243,Z 331.771,A -85,B 0,C 180,E1 -6583.47,E2 -6583.47} C_VEL
LIN {X 0,Y 490.671,Z 319.265,A -85,B 0,C 180,E1 -6584.039,E2 -6584.039} C_VEL
LIN {X 0,Y 490.965,Z 306.206,A -85,B 0,C 180,E1 -6584.453,E2 -6584.453} C_VEL
LIN {X 0,Y 491.179,Z 290.526,A -85,B 0,C 180,E1 -6584.738,E2 -6584.738} C_VEL
LIN {X 0,Y 491.604,Z 208.222,A -85,B 0,C 180,E1 -6585.978,E2 -6585.978} C_VEL
LIN {X 0,Y 489.328,Z 193.904,A -85,B 0,C 180,E1 -6586.306,E2 -6586.306} C_VEL
LIN {X 0,Y 489.796,Z 176.794,A -85,B 0,C 180,E1 -6589.269,E2 -6589.269} C_VEL
LIN {X 0,Y 490.426,Z 159.563,A -85,B 0,C 180,E1 -6592.317,E2 -6592.317} C_VEL
LIN {X 0,Y 489.079,Z 150.927,A -85,B 0,C 180,E1 -6593.949,E2 -6593.949} C_VEL
LIN {X 0,Y 488.74,Z 149.141,A -85,B 0,C 180,E1 -6594.362,E2 -6594.362} C_VEL
LIN {X 0,Y 488.676,Z 149.117,A -85,B 0,C 180,E1 -6597.4,E2 -6597.4} C_VEL
LIN {X 0,Y 488.648,Z 149.115,A -85,B 0,C 180,E1 -6600.35,E2 -6600.35} C_VEL
LIN {X 0,Y 488.705,Z 149.11,A -85,B 0,C 180,E1 -6603.478,E2 -6603.478} C_VEL
LIN {X 0,Y 488.641,Z 149.115,A -85,B 0,C 180,E1 -6606.347,E2 -6606.347} C_VEL
LIN {X 0,Y 488.676,Z 149.116,A -85,B 0,C 180,E1 -6609.255,E2 -6609.255} C_VEL
LIN {X 0,Y 488.659,Z 149.117,A -85,B 0,C 180,E1 -6611.593,E2 -6611.593} C_VEL
LIN {X 0,Y 488.687,Z 149.109,A -85,B 0,C 180,E1 -6614.802,E2 -6614.802} C_VEL
LIN {X 0,Y 488.639,Z 149.121,A -85,B 0,C 180,E1 -6617.468,E2 -6617.468} C_VEL
LIN {X 0,Y 488.695,Z 149.11,A -85,B 0,C 180,E1 -6619.672,E2 -6619.672} C_VEL
LIN {X 0,Y 488.65,Z 149.114,A -85,B 0,C 180,E1 -6622.838,E2 -6622.838} C_VEL
LIN {X 0,Y 488.707,Z 149.104,A -85,B 0,C 180,E1 -6625.885,E2 -6625.885} C_VEL
LIN {X 0,Y 488.655,Z 149.116,A -85,B 0,C 180,E1 -6628.817,E2 -6628.817} C_VEL
LIN {X 0,Y 488.681,Z 149.109,A -85,B 0,C 180,E1 -6631.667,E2 -6631.667} C_VEL
LIN {X 0,Y 488.649,Z 149.114,A -85,B 0,C 180,E1 -6634.438,E2 -6634.438} C_VEL
LIN {X 0,Y 488.708,Z 149.11,A -85,B 0,C 180,E1 -6637.152,E2 -6637.152} C_VEL
LIN {X 0,Y 488.706,Z 149.104,A -85,B 0,C 180,E1 -6639.809,E2 -6639.809} C_VEL
LIN {X 0,Y 488.694,Z 149.109,A -85,B 0,C 180,E1 -6642.422,E2 -6642.422} C_VEL
LIN {X 0,Y 488.739,Z 149.105,A -85,B 0,C 180,E1 -6644.999,E2 -6644.999} C_VEL
LIN {X 0,Y 488.79,Z 149.098,A -85,B 0,C 180,E1 -6648.387,E2 -6648.387} C_VEL
LIN {X 0,Y 488.768,Z 149.097,A -85,B 0,C 180,E1 -6651.732,E2 -6651.732} C_VEL
LIN {X 0,Y 488.819,Z 149.093,A -85,B 0,C 180,E1 -6654.223,E2 -6654.223} C_VEL
LIN {X 0,Y 488.933,Z 149.077,A -85,B 0,C 180,E1 -6657.528,E2 -6657.528} C_VEL
LIN {X 0,Y 488.897,Z 149.087,A -85,B 0,C 180,E1 -6660.823,E2 -6660.823} C_VEL
LIN {X 0,Y 488.931,Z 149.084,A -85,B 0,C 180,E1 -6662.471,E2 -6662.471} C_VEL
LIN {X 0,Y 488.818,Z 149.093,A -85,B 0,C 180,E1 -6665.776,E2 -6665.776} C_VEL
LIN {X 0,Y 488.758,Z 149.106,A -85,B 0,C 180,E1 -6668.267,E2 -6668.267} C_VEL
LIN {X 0,Y 488.768,Z 149.098,A -85,B 0,C 180,E1 -6671.613,E2 -6671.613} C_VEL
LIN {X 0,Y 488.742,Z 149.103,A -85,B 0,C 180,E1 -6675.001,E2 -6675.001} C_VEL
LIN {X 0,Y 488.729,Z 149.109,A -85,B 0,C 180,E1 -6678.443,E2 -6678.443} C_VEL
LIN {X 0,Y 488.693,Z 149.108,A -85,B 0,C 180,E1 -6681.071,E2 -6681.071} C_VEL
LIN {X 0,Y 488.655,Z 149.116,A -85,B 0,C 180,E1 -6683.747,E2 -6683.747} C_VEL
LIN {X 0,Y 488.682,Z 149.111,A -85,B 0,C 180,E1 -6686.922,E2 -6686.922} C_VEL
LIN {X 0,Y 488.703,Z 149.113,A -85,B 0,C 180,E1 -6690.22,E2 -6690.22} C_VEL
LIN {X 0,Y 488.76,Z 149.292,A -85,B 0,C 180,E1 -6691.968,E2 -6691.968} C_VEL
LIN {X 0,Y 489.917,Z 156.213,A -85,B 0,C 180,E1 -6693.364,E2 -6693.364} C_VEL
LIN {X 0,Y 489.556,Z 171.75,A -85,B 0,C 180,E1 -6696.271,E2 -6696.271} C_VEL
LIN {X 0,Y 489.396,Z 179.893,A -85,B 0,C 180,E1 -6697.745,E2 -6697.745} C_VEL
LIN {X 0,Y 491.799,Z 193.927,A -85,B 0,C 180,E1 -6698.078,E2 -6698.078} C_VEL
LIN {X 0,Y 491.088,Z 288.077,A -85,B 0,C 180,E1 -6699.515,E2 -6699.515} C_VEL
LIN {X 0,Y 490.817,Z 301.635,A -85,B 0,C 180,E1 -6699.9,E2 -6699.9} C_VEL
LIN {X 0,Y 490.522,Z 313.947,A -85,B 0,C 180,E1 -6700.419,E2 -6700.419} C_VEL
LIN {X 0,Y 490.123,Z 325.391,A -85,B 0,C 180,E1 -6701.067,E2 -6701.067} C_VEL
LIN {X 0,Y 489.696,Z 337.333,A -85,B 0,C 180,E1 -6701.939,E2 -6701.939} C_VEL
LIN {X 0,Y 489.273,Z 347.791,A -85,B 0,C 180,E1 -6702.9,E2 -6702.9} C_VEL
LIN {X 0,Y 488.87,Z 357.756,A -85,B 0,C 180,E1 -6704.047,E2 -6704.047} C_VEL
LIN {X 0,Y 488.527,Z 365.761,A -85,B 0,C 180,E1 -6705.179,E2 -6705.179} C_VEL
LIN {X 0,Y 488.437,Z 369.123,A -85,B 0,C 180,E1 -6705.734,E2 -6705.734} C_VEL
LIN {X 0,Y 487.67,Z 372.392,A -85,B 0,C 180,E1 -6706.306,E2 -6706.306} C_VEL
LIN {X 0,Y 484.659,Z 377.247,A -85,B 0,C 180,E1 -6707.263,E2 -6707.263} C_VEL
LIN {X 0,Y 481.669,Z 381.358,A -85,B 0,C 180,E1 -6708.276,E2 -6708.276} C_VEL
LIN {X 0,Y 480.947,Z 383.464,A -85,B 0,C 180,E1 -6708.93,E2 -6708.93} C_VEL
LIN {X 0,Y 480.839,Z 386.317,A -85,B 0,C 180,E1 -6709.978,E2 -6709.978} C_VEL
LIN {X 0,Y 480.735,Z 388.486,A -85,B 0,C 180,E1 -6711.053,E2 -6711.053} C_VEL
LIN {X 0,Y 480.696,Z 390.012,A -85,B 0,C 180,E1 -6712.139,E2 -6712.139} C_VEL
LIN {X 0,Y 480.651,Z 390.954,A -85,B 0,C 180,E1 -6713.532,E2 -6713.532} C_VEL
LIN {X 0,Y 480.673,Z 390.775,A -85,B 0,C 180,E1 -6714.963,E2 -6714.963} C_VEL
LIN {X 0,Y 480.712,Z 389.371,A -85,B 0,C 180,E1 -6716.442,E2 -6716.442} C_VEL
LIN {X 0,Y 480.835,Z 386.607,A -85,B 0,C 180,E1 -6717.966,E2 -6717.966} C_VEL
LIN {X 0,Y 480.937,Z 383.171,A -85,B 0,C 180,E1 -6719.24,E2 -6719.24} C_VEL
LIN {X 0,Y 481.109,Z 377.852,A -85,B 0,C 180,E1 -6720.703,E2 -6720.703} C_VEL
LIN {X 0,Y 481.337,Z 370.963,A -85,B 0,C 180,E1 -6722.147,E2 -6722.147} C_VEL
LIN {X 0,Y 481.592,Z 363.836,A -85,B 0,C 180,E1 -6723.338,E2 -6723.338} C_VEL
LIN {X 0,Y 481.968,Z 354.58,A -85,B 0,C 180,E1 -6724.584,E2 -6724.584} C_VEL
LIN {X 0,Y 482.425,Z 344.235,A -85,B 0,C 180,E1 -6725.699,E2 -6725.699} C_VEL
LIN {X 0,Y 482.876,Z 333.577,A -85,B 0,C 180,E1 -6726.622,E2 -6726.622} C_VEL
LIN {X 0,Y 483.259,Z 323.309,A -85,B 0,C 180,E1 -6727.334,E2 -6727.334} C_VEL
LIN {X 0,Y 483.632,Z 311.707,A -85,B 0,C 180,E1 -6727.964,E2 -6727.964} C_VEL
LIN {X 0,Y 484.005,Z 298.635,A -85,B 0,C 180,E1 -6728.486,E2 -6728.486} C_VEL
LIN {X 0,Y 484.231,Z 286.375,A -85,B 0,C 180,E1 -6728.81,E2 -6728.81} C_VEL
LIN {X 0,Y 484.749,Z 193.484,A -85,B 0,C 180,E1 -6730.233,E2 -6730.233} C_VEL
LIN {X 0,Y 482.386,Z 180.23,A -85,B 0,C 180,E1 -6730.545,E2 -6730.545} C_VEL
LIN {X 0,Y 482.612,Z 172.634,A -85,B 0,C 180,E1 -6731.975,E2 -6731.975} C_VEL
LIN {X 0,Y 483.115,Z 158.233,A -85,B 0,C 180,E1 -6734.821,E2 -6734.821} C_VEL
LIN {X 0,Y 481.751,Z 150.051,A -85,B 0,C 180,E1 -6736.583,E2 -6736.583} C_VEL
LIN {X 0,Y 481.704,Z 149.982,A -85,B 0,C 180,E1 -6739.068,E2 -6739.068} C_VEL
LIN {X 0,Y 481.825,Z 149.964,A -85,B 0,C 180,E1 -6742.458,E2 -6742.458} C_VEL
LIN {X 0,Y 481.778,Z 149.968,A -85,B 0,C 180,E1 -6744.98,E2 -6744.98} C_VEL
LIN {X 0,Y 481.924,Z 149.954,A -85,B 0,C 180,E1 -6747.493,E2 -6747.493} C_VEL
LIN {X 0,Y 481.937,Z 149.953,A -85,B 0,C 180,E1 -6750.001,E2 -6750.001} C_VEL
LIN {X 0,Y 481.925,Z 149.95,A -85,B 0,C 180,E1 -6752.508,E2 -6752.508} C_VEL
LIN {X 0,Y 481.805,Z 149.97,A -85,B 0,C 180,E1 -6755.861,E2 -6755.861} C_VEL
LIN {X 0,Y 481.739,Z 149.973,A -85,B 0,C 180,E1 -6758.389,E2 -6758.389} C_VEL
LIN {X 0,Y 481.749,Z 149.976,A -85,B 0,C 180,E1 -6761.786,E2 -6761.786} C_VEL
LIN {X 0,Y 481.741,Z 149.978,A -85,B 0,C 180,E1 -6765.225,E2 -6765.225} C_VEL
LIN {X 0,Y 481.707,Z 149.978,A -85,B 0,C 180,E1 -6768.723,E2 -6768.723} C_VEL
LIN {X 0,Y 481.645,Z 149.991,A -85,B 0,C 180,E1 -6771.395,E2 -6771.395} C_VEL
LIN {X 0,Y 481.657,Z 149.983,A -85,B 0,C 180,E1 -6774.115,E2 -6774.115} C_VEL
LIN {X 0,Y 481.745,Z 149.98,A -85,B 0,C 180,E1 -6777.139,E2 -6777.139} C_VEL
LIN {X 0,Y 481.677,Z 149.982,A -85,B 0,C 180,E1 -6779.742,E2 -6779.742} C_VEL
LIN {X 0,Y 481.669,Z 149.985,A -85,B 0,C 180,E1 -6782.675,E2 -6782.675} C_VEL
LIN {X 0,Y 481.635,Z 149.986,A -85,B 0,C 180,E1 -6785.71,E2 -6785.71} C_VEL
LIN {X 0,Y 481.667,Z 149.99,A -85,B 0,C 180,E1 -6788.86,E2 -6788.86} C_VEL
LIN {X 0,Y 481.651,Z 149.984,A -85,B 0,C 180,E1 -6791.913,E2 -6791.913} C_VEL
LIN {X 0,Y 481.654,Z 149.987,A -85,B 0,C 180,E1 -6794.458,E2 -6794.458} C_VEL
LIN {X 0,Y 481.642,Z 149.985,A -85,B 0,C 180,E1 -6797.839,E2 -6797.839} C_VEL
LIN {X 0,Y 481.658,Z 149.991,A -85,B 0,C 180,E1 -6800.655,E2 -6800.655} C_VEL
LIN {X 0,Y 481.62,Z 149.988,A -85,B 0,C 180,E1 -6803.378,E2 -6803.378} C_VEL
LIN {X 0,Y 481.693,Z 149.984,A -85,B 0,C 180,E1 -6806.329,E2 -6806.329} C_VEL
LIN {X 0,Y 481.648,Z 149.984,A -85,B 0,C 180,E1 -6809.418,E2 -6809.418} C_VEL
LIN {X 0,Y 481.666,Z 149.987,A -85,B 0,C 180,E1 -6812.166,E2 -6812.166} C_VEL
LIN {X 0,Y 481.678,Z 149.981,A -85,B 0,C 180,E1 -6814.968,E2 -6814.968} C_VEL
LIN {X 0,Y 481.647,Z 149.986,A -85,B 0,C 180,E1 -6817.705,E2 -6817.705} C_VEL
LIN {X 0,Y 481.701,Z 149.983,A -85,B 0,C 180,E1 -6820.393,E2 -6820.393} C_VEL
LIN {X 0,Y 481.671,Z 149.981,A -85,B 0,C 180,E1 -6823.034,E2 -6823.034} C_VEL
LIN {X 0,Y 481.68,Z 149.983,A -85,B 0,C 180,E1 -6825.639,E2 -6825.639} C_VEL
LIN {X 0,Y 481.75,Z 149.977,A -85,B 0,C 180,E1 -6828.215,E2 -6828.215} C_VEL
LIN {X 0,Y 481.721,Z 149.979,A -85,B 0,C 180,E1 -6831.611,E2 -6831.611} C_VEL
LIN {X 0,Y 481.775,Z 149.974,A -85,B 0,C 180,E1 -6834.139,E2 -6834.139} C_VEL
LIN {X 0,Y 481.907,Z 149.956,A -85,B 0,C 180,E1 -6837.493,E2 -6837.493} C_VEL
LIN {X 0,Y 481.909,Z 149.957,A -85,B 0,C 180,E1 -6840,E2 -6840} C_VEL
LIN {X 0,Y 481.915,Z 149.951,A -85,B 0,C 180,E1 -6842.508,E2 -6842.508} C_VEL
LIN {X 0,Y 481.765,Z 149.975,A -85,B 0,C 180,E1 -6845.861,E2 -6845.861} C_VEL
LIN {X 0,Y 481.718,Z 149.976,A -85,B 0,C 180,E1 -6848.389,E2 -6848.389} C_VEL
LIN {X 0,Y 481.75,Z 149.976,A -85,B 0,C 180,E1 -6851.785,E2 -6851.785} C_VEL
LIN {X 0,Y 481.737,Z 149.978,A -85,B 0,C 180,E1 -6855.225,E2 -6855.225} C_VEL
LIN {X 0,Y 481.705,Z 149.978,A -85,B 0,C 180,E1 -6858.722,E2 -6858.722} C_VEL
LIN {X 0,Y 481.644,Z 149.992,A -85,B 0,C 180,E1 -6861.395,E2 -6861.395} C_VEL
LIN {X 0,Y 481.643,Z 149.985,A -85,B 0,C 180,E1 -6864.115,E2 -6864.115} C_VEL
LIN {X 0,Y 481.643,Z 149.992,A -85,B 0,C 180,E1 -6867.115,E2 -6867.115} C_VEL
LIN {X 0,Y 481.6,Z 149.991,A -85,B 0,C 180,E1 -6869.747,E2 -6869.747} C_VEL
LIN {X 0,Y 481.635,Z 149.989,A -85,B 0,C 180,E1 -6872.677,E2 -6872.677} C_VEL
LIN {X 0,Y 481.649,Z 149.99,A -85,B 0,C 180,E1 -6875.202,E2 -6875.202} C_VEL
LIN {X 0,Y 481.63,Z 149.986,A -85,B 0,C 180,E1 -6878.003,E2 -6878.003} C_VEL
LIN {X 0,Y 481.605,Z 149.996,A -85,B 0,C 180,E1 -6881.048,E2 -6881.048} C_VEL
LIN {X 0,Y 481.652,Z 149.987,A -85,B 0,C 180,E1 -6884.459,E2 -6884.459} C_VEL
LIN {X 0,Y 481.614,Z 149.996,A -85,B 0,C 180,E1 -6886.856,E2 -6886.856} C_VEL
LIN {X 0,Y 481.629,Z 149.988,A -85,B 0,C 180,E1 -6890.054,E2 -6890.054} C_VEL
LIN {X 0,Y 481.588,Z 149.993,A -85,B 0,C 180,E1 -6893.249,E2 -6893.249} C_VEL
LIN {X 0,Y 481.618,Z 149.993,A -85,B 0,C 180,E1 -6896.322,E2 -6896.322} C_VEL
LIN {X 0,Y 481.613,Z 149.991,A -85,B 0,C 180,E1 -6899.426,E2 -6899.426} C_VEL
LIN {X 0,Y 481.644,Z 149.992,A -85,B 0,C 180,E1 -6902.164,E2 -6902.164} C_VEL
LIN {X 0,Y 481.692,Z 150.188,A -85,B 0,C 180,E1 -6905.428,E2 -6905.428} C_VEL
LIN {X 0,Y 483.489,Z 159.89,A -85,B 0,C 180,E1 -6907.343,E2 -6907.343} C_VEL
LIN {X 0,Y 483.109,Z 170.843,A -85,B 0,C 180,E1 -6909.342,E2 -6909.342} C_VEL
LIN {X 0,Y 482.504,Z 187.853,A -85,B 0,C 180,E1 -6912.407,E2 -6912.407} C_VEL
LIN {X 0,Y 482.334,Z 193.982,A -85,B 0,C 180,E1 -6913.473,E2 -6913.473} C_VEL
LIN {X 0,Y 482.965,Z 198.329,A -85,B 0,C 180,E1 -6913.603,E2 -6913.603} C_VEL
LIN {X 0,Y 484.834,Z 210.242,A -85,B 0,C 180,E1 -6913.849,E2 -6913.849} C_VEL
LIN {X 0,Y 484.216,Z 302.173,A -85,B 0,C 180,E1 -6915.258,E2 -6915.258} C_VEL
LIN {X 0,Y 483.897,Z 315.287,A -85,B 0,C 180,E1 -6915.624,E2 -6915.624} C_VEL
LIN {X 0,Y 483.493,Z 327.381,A -85,B 0,C 180,E1 -6916.122,E2 -6916.122} C_VEL
LIN {X 0,Y 483.13,Z 338.805,A -85,B 0,C 180,E1 -6916.755,E2 -6916.755} C_VEL
LIN {X 0,Y 482.684,Z 350.54,A -85,B 0,C 180,E1 -6917.598,E2 -6917.598} C_VEL
LIN {X 0,Y 482.278,Z 361.081,A -85,B 0,C 180,E1 -6918.547,E2 -6918.547} C_VEL
LIN {X 0,Y 481.856,Z 369.693,A -85,B 0,C 180,E1 -6919.495,E2 -6919.495} C_VEL
LIN {X 0,Y 481.53,Z 377.633,A -85,B 0,C 180,E1 -6920.549,E2 -6920.549} C_VEL
LIN {X 0,Y 481.241,Z 385.391,A -85,B 0,C 180,E1 -6921.813,E2 -6921.813} C_VEL
LIN {X 0,Y 481.004,Z 392.518,A -85,B 0,C 180,E1 -6923.287,E2 -6923.287} C_VEL
LIN {X 0,Y 480.961,Z 397.264,A -85,B 0,C 180,E1 -6924.549,E2 -6924.549} C_VEL
LIN {X 0,Y 480.828,Z 400.887,A -85,B 0,C 180,E1 -6925.808,E2 -6925.808} C_VEL
LIN {X 0,Y 480.871,Z 402.759,A -85,B 0,C 180,E1 -6926.648,E2 -6926.648} C_VEL
LIN {X 0,Y 480.804,Z 404.16,A -85,B 0,C 180,E1 -6927.486,E2 -6927.486} C_VEL
LIN {X 0,Y 480.79,Z 405.158,A -85,B 0,C 180,E1 -6928.324,E2 -6928.324} C_VEL
LIN {X 0,Y 480.76,Z 405.767,A -85,B 0,C 180,E1 -6929.162,E2 -6929.162} C_VEL
LIN {X 0,Y 480.744,Z 405.984,A -85,B 0,C 180,E1 -6929.999,E2 -6929.999} C_VEL
LIN {X 0,Y 480.76,Z 405.766,A -85,B 0,C 180,E1 -6930.837,E2 -6930.837} C_VEL
LIN {X 0,Y 480.79,Z 405.156,A -85,B 0,C 180,E1 -6931.674,E2 -6931.674} C_VEL
LIN {X 0,Y 480.87,Z 402.755,A -85,B 0,C 180,E1 -6933.351,E2 -6933.351} C_VEL
LIN {X 0,Y 480.839,Z 399.807,A -85,B 0,C 180,E1 -6934.61,E2 -6934.61} C_VEL
LIN {X 0,Y 480.96,Z 395.819,A -85,B 0,C 180,E1 -6935.87,E2 -6935.87} C_VEL
LIN {X 0,Y 481.11,Z 389.68,A -85,B 0,C 180,E1 -6937.343,E2 -6937.343} C_VEL
LIN {X 0,Y 481.323,Z 382.974,A -85,B 0,C 180,E1 -6938.606,E2 -6938.606} C_VEL
LIN {X 0,Y 481.672,Z 374.654,A -85,B 0,C 180,E1 -6939.871,E2 -6939.871} C_VEL
LIN {X 0,Y 482.02,Z 366.107,A -85,B 0,C 180,E1 -6940.925,E2 -6940.925} C_VEL
LIN {X 0,Y 482.477,Z 355.553,A -85,B 0,C 180,E1 -6941.979,E2 -6941.979} C_VEL
LIN {X 0,Y 482.903,Z 343.968,A -85,B 0,C 180,E1 -6942.907,E2 -6942.907} C_VEL
LIN {X 0,Y 483.299,Z 333.629,A -85,B 0,C 180,E1 -6943.56,E2 -6943.56} C_VEL
LIN {X 0,Y 483.721,Z 321.757,A -85,B 0,C 180,E1 -6944.138,E2 -6944.138} C_VEL
LIN {X 0,Y 484.066,Z 308.07,A -85,B 0,C 180,E1 -6944.61,E2 -6944.61} C_VEL
LIN {X 0,Y 484.289,Z 295.767,A -85,B 0,C 180,E1 -6944.872,E2 -6944.872} C_VEL
LIN {X 0,Y 484.839,Z 209.335,A -85,B 0,C 180,E1 -6946.192,E2 -6946.192} C_VEL
LIN {X 0,Y 482.357,Z 193.998,A -85,B 0,C 180,E1 -6946.536,E2 -6946.536} C_VEL
LIN {X 0,Y 482.691,Z 182.848,A -85,B 0,C 180,E1 -6948.461,E2 -6948.461} C_VEL
LIN {X 0,Y 483.426,Z 163.153,A -85,B 0,C 180,E1 -6951.986,E2 -6951.986} C_VEL
LIN {X 0,Y 483.212,Z 158.25,A -85,B 0,C 180,E1 -6952.895,E2 -6952.895} C_VEL
LIN {X 0,Y 481.69,Z 150.122,A -85,B 0,C 180,E1 -6954.512,E2 -6954.512} C_VEL
LIN {X 0,Y 481.64,Z 149.992,A -85,B 0,C 180,E1 -6957.834,E2 -6957.834} C_VEL
LIN {X 0,Y 481.606,Z 149.993,A -85,B 0,C 180,E1 -6960.712,E2 -6960.712} C_VEL
LIN {X 0,Y 481.671,Z 149.988,A -85,B 0,C 180,E1 -6963.728,E2 -6963.728} C_VEL
LIN {X 0,Y 481.598,Z 149.993,A -85,B 0,C 180,E1 -6966.748,E2 -6966.748} C_VEL
LIN {X 0,Y 481.647,Z 149.987,A -85,B 0,C 180,E1 -6969.941,E2 -6969.941} C_VEL
LIN {X 0,Y 481.606,Z 149.999,A -85,B 0,C 180,E1 -6973.301,E2 -6973.301} C_VEL
LIN {X 0,Y 481.64,Z 149.99,A -85,B 0,C 180,E1 -6975.641,E2 -6975.641} C_VEL
LIN {X 0,Y 481.614,Z 149.994,A -85,B 0,C 180,E1 -6978.953,E2 -6978.953} C_VEL
LIN {X 0,Y 481.624,Z 149.986,A -85,B 0,C 180,E1 -6981.995,E2 -6981.995} C_VEL
LIN {X 0,Y 481.671,Z 149.985,A -85,B 0,C 180,E1 -6985.316,E2 -6985.316} C_VEL
LIN {X 0,Y 481.613,Z 149.989,A -85,B 0,C 180,E1 -6988.309,E2 -6988.309} C_VEL
LIN {X 0,Y 481.642,Z 149.99,A -85,B 0,C 180,E1 -6991.214,E2 -6991.214} C_VEL
LIN {X 0,Y 481.617,Z 149.988,A -85,B 0,C 180,E1 -6994.038,E2 -6994.038} C_VEL
LIN {X 0,Y 481.641,Z 149.989,A -85,B 0,C 180,E1 -6996.817,E2 -6996.817} C_VEL
LIN {X 0,Y 481.68,Z 149.981,A -85,B 0,C 180,E1 -6999.502,E2 -6999.502} C_VEL
LIN {X 0,Y 481.673,Z 149.981,A -85,B 0,C 180,E1 -7002.157,E2 -7002.157} C_VEL
LIN {X 0,Y 481.724,Z 149.978,A -85,B 0,C 180,E1 -7004.775,E2 -7004.775} C_VEL
LIN {X 0,Y 481.736,Z 149.975,A -85,B 0,C 180,E1 -7008.214,E2 -7008.214} C_VEL
LIN {X 0,Y 481.723,Z 149.975,A -85,B 0,C 180,E1 -7011.611,E2 -7011.611} C_VEL
LIN {X 0,Y 481.78,Z 149.969,A -85,B 0,C 180,E1 -7014.139,E2 -7014.139} C_VEL
LIN {X 0,Y 481.9,Z 149.953,A -85,B 0,C 180,E1 -7017.492,E2 -7017.492} C_VEL
LIN {X 0,Y 481.85,Z 149.964,A -85,B 0,C 180,E1 -7020.835,E2 -7020.835} C_VEL
LIN {X 0,Y 481.897,Z 149.96,A -85,B 0,C 180,E1 -7022.507,E2 -7022.507} C_VEL
LIN {X 0,Y 481.779,Z 149.97,A -85,B 0,C 180,E1 -7025.86,E2 -7025.86} C_VEL
LIN {X 0,Y 481.713,Z 149.984,A -85,B 0,C 180,E1 -7028.389,E2 -7028.389} C_VEL
LIN {X 0,Y 481.719,Z 149.977,A -85,B 0,C 180,E1 -7031.785,E2 -7031.785} C_VEL
LIN {X 0,Y 481.725,Z 149.976,A -85,B 0,C 180,E1 -7035.224,E2 -7035.224} C_VEL
LIN {X 0,Y 481.691,Z 149.983,A -85,B 0,C 180,E1 -7038.722,E2 -7038.722} C_VEL
LIN {X 0,Y 481.631,Z 149.988,A -85,B 0,C 180,E1 -7041.395,E2 -7041.395} C_VEL
LIN {X 0,Y 481.634,Z 149.995,A -85,B 0,C 180,E1 -7044.115,E2 -7044.115} C_VEL
LIN {X 0,Y 481.636,Z 149.988,A -85,B 0,C 180,E1 -7047.117,E2 -7047.117} C_VEL
LIN {X 0,Y 481.651,Z 149.99,A -85,B 0,C 180,E1 -7049.743,E2 -7049.743} C_VEL
LIN {X 0,Y 481.721,Z 150.134,A -85,B 0,C 180,E1 -7051.772,E2 -7051.772} C_VEL
LIN {X 0,Y 482.982,Z 157.693,A -85,B 0,C 180,E1 -7053.319,E2 -7053.319} C_VEL
LIN {X 0,Y 482.597,Z 172.584,A -85,B 0,C 180,E1 -7056.142,E2 -7056.142} C_VEL
LIN {X 0,Y 482.426,Z 179.981,A -85,B 0,C 180,E1 -7057.495,E2 -7057.495} C_VEL
LIN {X 0,Y 483.997,Z 188.795,A -85,B 0,C 180,E1 -7057.724,E2 -7057.724} C_VEL
LIN {X 0,Y 484.993,Z 195.063,A -85,B 0,C 180,E1 -7057.859,E2 -7057.859} C_VEL
LIN {X 0,Y 484.222,Z 287.406,A -85,B 0,C 180,E1 -7059.284,E2 -7059.284} C_VEL
LIN {X 0,Y 483.987,Z 300.644,A -85,B 0,C 180,E1 -7059.656,E2 -7059.656} C_VEL
LIN {X 0,Y 483.652,Z 312.633,A -85,B 0,C 180,E1 -7060.152,E2 -7060.152} C_VEL
LIN {X 0,Y 483.272,Z 324.19,A -85,B 0,C 180,E1 -7060.791,E2 -7060.791} C_VEL
LIN {X 0,Y 482.831,Z 335.484,A -85,B 0,C 180,E1 -7061.602,E2 -7061.602} C_VEL
LIN {X 0,Y 482.408,Z 346.116,A -85,B 0,C 180,E1 -7062.558,E2 -7062.558} C_VEL
LIN {X 0,Y 481.953,Z 355.988,A -85,B 0,C 180,E1 -7063.657,E2 -7063.657} C_VEL
LIN {X 0,Y 481.616,Z 363.753,A -85,B 0,C 180,E1 -7064.719,E2 -7064.719} C_VEL
LIN {X 0,Y 481.316,Z 370.941,A -85,B 0,C 180,E1 -7065.919,E2 -7065.919} C_VEL
LIN {X 0,Y 481.108,Z 377.753,A -85,B 0,C 180,E1 -7067.346,E2 -7067.346} C_VEL
LIN {X 0,Y 480.988,Z 382.195,A -85,B 0,C 180,E1 -7068.532,E2 -7068.532} C_VEL
LIN {X 0,Y 480.947,Z 383.464,A -85,B 0,C 180,E1 -7068.93,E2 -7068.93} C_VEL
LIN {X 0,Y 480.22,Z 385.377,A -85,B 0,C 180,E1 -7069.593,E2 -7069.593} C_VEL
LIN {X 0,Y 477.225,Z 387.943,A -85,B 0,C 180,E1 -7070.683,E2 -7070.683} C_VEL
LIN {X 0,Y 474.721,Z 389.44,A -85,B 0,C 180,E1 -7071.575,E2 -7071.575} C_VEL
LIN {X 0,Y 473.654,Z 390.278,A -85,B 0,C 180,E1 -7072.272,E2 -7072.272} C_VEL
LIN {X 0,Y 473.572,Z 390.497,A -85,B 0,C 180,E1 -7072.508,E2 -7072.508} C_VEL
LIN {X 0,Y 473.554,Z 391.076,A -85,B 0,C 180,E1 -7073.586,E2 -7073.586} C_VEL
LIN {X 0,Y 473.591,Z 391.027,A -85,B 0,C 180,E1 -7074.704,E2 -7074.704} C_VEL
LIN {X 0,Y 473.623,Z 389.847,A -85,B 0,C 180,E1 -7076.198,E2 -7076.198} C_VEL
LIN {X 0,Y 473.717,Z 387.305,A -85,B 0,C 180,E1 -7077.74,E2 -7077.74} C_VEL
LIN {X 0,Y 473.852,Z 383.196,A -85,B 0,C 180,E1 -7079.342,E2 -7079.342} C_VEL
LIN {X 0,Y 474.018,Z 378.334,A -85,B 0,C 180,E1 -7080.709,E2 -7080.709} C_VEL
LIN {X 0,Y 474.26,Z 371.525,A -85,B 0,C 180,E1 -7082.175,E2 -7082.175} C_VEL
LIN {X 0,Y 474.535,Z 364.484,A -85,B 0,C 180,E1 -7083.385,E2 -7083.385} C_VEL
LIN {X 0,Y 474.913,Z 355.895,A -85,B 0,C 180,E1 -7084.587,E2 -7084.587} C_VEL
LIN {X 0,Y 475.353,Z 346.433,A -85,B 0,C 180,E1 -7085.656,E2 -7085.656} C_VEL
LIN {X 0,Y 475.834,Z 335.959,A -85,B 0,C 180,E1 -7086.614,E2 -7086.614} C_VEL
LIN {X 0,Y 476.307,Z 324.662,A -85,B 0,C 180,E1 -7087.442,E2 -7087.442} C_VEL
LIN {X 0,Y 476.701,Z 312.991,A -85,B 0,C 180,E1 -7088.105,E2 -7088.105} C_VEL
LIN {X 0,Y 477.023,Z 300.094,A -85,B 0,C 180,E1 -7088.644,E2 -7088.644} C_VEL
LIN {X 0,Y 477.354,Z 287.382,A -85,B 0,C 180,E1 -7088.999,E2 -7088.999} C_VEL
LIN {X 0,Y 477.988,Z 194.769,A -85,B 0,C 180,E1 -7090.446,E2 -7090.446} C_VEL
LIN {X 0,Y 475.426,Z 180.382,A -85,B 0,C 180,E1 -7090.785,E2 -7090.785} C_VEL
LIN {X 0,Y 475.512,Z 176.417,A -85,B 0,C 180,E1 -7091.506,E2 -7091.506} C_VEL
LIN {X 0,Y 476.163,Z 159.859,A -85,B 0,C 180,E1 -7094.813,E2 -7094.813} C_VEL
LIN {X 0,Y 474.706,Z 150.98,A -85,B 0,C 180,E1 -7096.735,E2 -7096.735} C_VEL
LIN {X 0,Y 474.677,Z 150.859,A -85,B 0,C 180,E1 -7099.767,E2 -7099.767} C_VEL
LIN {X 0,Y 474.795,Z 150.838,A -85,B 0,C 180,E1 -7102.629,E2 -7102.629} C_VEL
LIN {X 0,Y 474.749,Z 150.844,A -85,B 0,C 180,E1 -7104.905,E2 -7104.905} C_VEL
LIN {X 0,Y 474.89,Z 150.83,A -85,B 0,C 180,E1 -7107.456,E2 -7107.456} C_VEL
LIN {X 0,Y 474.908,Z 150.828,A -85,B 0,C 180,E1 -7110.001,E2 -7110.001} C_VEL
LIN {X 0,Y 474.891,Z 150.826,A -85,B 0,C 180,E1 -7112.545,E2 -7112.545} C_VEL
LIN {X 0,Y 474.768,Z 150.845,A -85,B 0,C 180,E1 -7115.949,E2 -7115.949} C_VEL
LIN {X 0,Y 474.711,Z 150.848,A -85,B 0,C 180,E1 -7118.515,E2 -7118.515} C_VEL
LIN {X 0,Y 474.703,Z 150.852,A -85,B 0,C 180,E1 -7121.963,E2 -7121.963} C_VEL
LIN {X 0,Y 474.698,Z 150.858,A -85,B 0,C 180,E1 -7125.456,E2 -7125.456} C_VEL
LIN {X 0,Y 474.662,Z 150.858,A -85,B 0,C 180,E1 -7129.011,E2 -7129.011} C_VEL
LIN {X 0,Y 474.587,Z 150.866,A -85,B 0,C 180,E1 -7131.73,E2 -7131.73} C_VEL
LIN {X 0,Y 474.638,Z 150.858,A -85,B 0,C 180,E1 -7134.495,E2 -7134.495} C_VEL
LIN {X 0,Y 474.679,Z 150.858,A -85,B 0,C 180,E1 -7137.335,E2 -7137.335} C_VEL
LIN {X 0,Y 474.603,Z 150.862,A -85,B 0,C 180,E1 -7140.231,E2 -7140.231} C_VEL
LIN {X 0,Y 474.624,Z 150.865,A -85,B 0,C 180,E1 -7143.222,E2 -7143.222} C_VEL
LIN {X 0,Y 474.587,Z 150.865,A -85,B 0,C 180,E1 -7146.324,E2 -7146.324} C_VEL
LIN {X 0,Y 474.615,Z 150.861,A -85,B 0,C 180,E1 -7149.646,E2 -7149.646} C_VEL
LIN {X 0,Y 474.613,Z 150.867,A -85,B 0,C 180,E1 -7152.935,E2 -7152.935} C_VEL
LIN {X 0,Y 474.602,Z 150.862,A -85,B 0,C 180,E1 -7155.895,E2 -7155.895} C_VEL
LIN {X 0,Y 474.621,Z 150.863,A -85,B 0,C 180,E1 -7159.042,E2 -7159.042} C_VEL
LIN {X 0,Y 474.606,Z 150.861,A -85,B 0,C 180,E1 -7161.705,E2 -7161.705} C_VEL
LIN {X 0,Y 474.621,Z 150.865,A -85,B 0,C 180,E1 -7164.726,E2 -7164.726} C_VEL
LIN {X 0,Y 474.634,Z 150.859,A -85,B 0,C 180,E1 -7167.788,E2 -7167.788} C_VEL
LIN {X 0,Y 474.605,Z 150.864,A -85,B 0,C 180,E1 -7170.889,E2 -7170.889} C_VEL
LIN {X 0,Y 474.613,Z 150.861,A -85,B 0,C 180,E1 -7173.626,E2 -7173.626} C_VEL
LIN {X 0,Y 474.634,Z 150.862,A -85,B 0,C 180,E1 -7176.642,E2 -7176.642} C_VEL
LIN {X 0,Y 474.652,Z 150.862,A -85,B 0,C 180,E1 -7180.09,E2 -7180.09} C_VEL
LIN {X 0,Y 474.632,Z 150.859,A -85,B 0,C 180,E1 -7182.774,E2 -7182.774} C_VEL
LIN {X 0,Y 474.64,Z 150.858,A -85,B 0,C 180,E1 -7185.421,E2 -7185.421} C_VEL
LIN {X 0,Y 474.704,Z 150.858,A -85,B 0,C 180,E1 -7188.038,E2 -7188.038} C_VEL
LIN {X 0,Y 474.696,Z 150.852,A -85,B 0,C 180,E1 -7191.486,E2 -7191.486} C_VEL
LIN {X 0,Y 474.738,Z 150.851,A -85,B 0,C 180,E1 -7194.052,E2 -7194.052} C_VEL
LIN {X 0,Y 474.872,Z 150.831,A -85,B 0,C 180,E1 -7197.456,E2 -7197.456} C_VEL
LIN {X 0,Y 474.878,Z 150.833,A -85,B 0,C 180,E1 -7200,E2 -7200} C_VEL
LIN {X 0,Y 474.881,Z 150.827,A -85,B 0,C 180,E1 -7202.545,E2 -7202.545} C_VEL
LIN {X 0,Y 474.729,Z 150.85,A -85,B 0,C 180,E1 -7205.949,E2 -7205.949} C_VEL
LIN {X 0,Y 474.667,Z 150.854,A -85,B 0,C 180,E1 -7208.515,E2 -7208.515} C_VEL
LIN {X 0,Y 474.704,Z 150.852,A -85,B 0,C 180,E1 -7211.963,E2 -7211.963} C_VEL
LIN {X 0,Y 474.68,Z 150.856,A -85,B 0,C 180,E1 -7215.767,E2 -7215.767} C_VEL
LIN {X 0,Y 474.659,Z 150.858,A -85,B 0,C 180,E1 -7219.011,E2 -7219.011} C_VEL
LIN {X 0,Y 474.587,Z 150.867,A -85,B 0,C 180,E1 -7221.729,E2 -7221.729} C_VEL
LIN {X 0,Y 474.621,Z 150.86,A -85,B 0,C 180,E1 -7224.495,E2 -7224.495} C_VEL
LIN {X 0,Y 474.594,Z 150.869,A -85,B 0,C 180,E1 -7227.327,E2 -7227.327} C_VEL
LIN {X 0,Y 474.55,Z 150.868,A -85,B 0,C 180,E1 -7230.234,E2 -7230.234} C_VEL
LIN {X 0,Y 474.609,Z 150.867,A -85,B 0,C 180,E1 -7233.223,E2 -7233.223} C_VEL
LIN {X 0,Y 474.571,Z 150.867,A -85,B 0,C 180,E1 -7236.325,E2 -7236.325} C_VEL
LIN {X 0,Y 474.601,Z 150.863,A -85,B 0,C 180,E1 -7239.551,E2 -7239.551} C_VEL
LIN {X 0,Y 474.567,Z 150.873,A -85,B 0,C 180,E1 -7242.94,E2 -7242.94} C_VEL
LIN {X 0,Y 474.582,Z 150.864,A -85,B 0,C 180,E1 -7245.891,E2 -7245.891} C_VEL
LIN {X 0,Y 474.582,Z 150.868,A -85,B 0,C 180,E1 -7249.048,E2 -7249.048} C_VEL
LIN {X 0,Y 474.583,Z 150.864,A -85,B 0,C 180,E1 -7251.709,E2 -7251.709} C_VEL
LIN {X 0,Y 474.563,Z 150.873,A -85,B 0,C 180,E1 -7254.72,E2 -7254.72} C_VEL
LIN {X 0,Y 474.611,Z 150.861,A -85,B 0,C 180,E1 -7257.785,E2 -7257.785} C_VEL
LIN {X 0,Y 474.578,Z 150.871,A -85,B 0,C 180,E1 -7260.895,E2 -7260.895} C_VEL
LIN {X 0,Y 474.575,Z 150.868,A -85,B 0,C 180,E1 -7263.623,E2 -7263.623} C_VEL
LIN {X 0,Y 474.662,Z 151.011,A -85,B 0,C 180,E1 -7265.215,E2 -7265.215} C_VEL
LIN {X 0,Y 476.516,Z 160.974,A -85,B 0,C 180,E1 -7267.222,E2 -7267.222} C_VEL
LIN {X 0,Y 476.214,Z 170.71,A -85,B 0,C 180,E1 -7269.029,E2 -7269.029} C_VEL
LIN {X 0,Y 475.518,Z 187.728,A -85,B 0,C 180,E1 -7272.14,E2 -7272.14} C_VEL
LIN {X 0,Y 475.398,Z 194.094,A -85,B 0,C 180,E1 -7273.246,E2 -7273.246} C_VEL
LIN {X 0,Y 478.021,Z 211.288,A -85,B 0,C 180,E1 -7273.634,E2 -7273.634} C_VEL
LIN {X 0,Y 477.353,Z 301.716,A -85,B 0,C 180,E1 -7275.041,E2 -7275.041} C_VEL
LIN {X 0,Y 476.989,Z 314.942,A -85,B 0,C 180,E1 -7275.412,E2 -7275.412} C_VEL
LIN {X 0,Y 476.544,Z 328.221,A -85,B 0,C 180,E1 -7275.97,E2 -7275.97} C_VEL
LIN {X 0,Y 476.12,Z 340.65,A -85,B 0,C 180,E1 -7276.697,E2 -7276.697} C_VEL
LIN {X 0,Y 475.695,Z 351.367,A -85,B 0,C 180,E1 -7277.498,E2 -7277.498} C_VEL
LIN {X 0,Y 475.248,Z 361.97,A -85,B 0,C 180,E1 -7278.483,E2 -7278.483} C_VEL
LIN {X 0,Y 474.759,Z 371.241,A -85,B 0,C 180,E1 -7279.551,E2 -7279.551} C_VEL
LIN {X 0,Y 474.388,Z 380.246,A -85,B 0,C 180,E1 -7280.835,E2 -7280.835} C_VEL
LIN {X 0,Y 474.101,Z 387.495,A -85,B 0,C 180,E1 -7282.118,E2 -7282.118} C_VEL
LIN {X 0,Y 473.885,Z 393.829,A -85,B 0,C 180,E1 -7283.542,E2 -7283.542} C_VEL
LIN {X 0,Y 473.837,Z 398.461,A -85,B 0,C 180,E1 -7284.894,E2 -7284.894} C_VEL
LIN {X 0,Y 473.735,Z 400.766,A -85,B 0,C 180,E1 -7285.745,E2 -7285.745} C_VEL
LIN {X 0,Y 473.765,Z 402.64,A -85,B 0,C 180,E1 -7286.597,E2 -7286.597} C_VEL
LIN {X 0,Y 473.723,Z 404.045,A -85,B 0,C 180,E1 -7287.448,E2 -7287.448} C_VEL
LIN {X 0,Y 473.689,Z 405.655,A -85,B 0,C 180,E1 -7289.149,E2 -7289.149} C_VEL
LIN {X 0,Y 473.67,Z 405.874,A -85,B 0,C 180,E1 -7289.999,E2 -7289.999} C_VEL
LIN {X 0,Y 473.688,Z 405.658,A -85,B 0,C 180,E1 -7290.849,E2 -7290.849} C_VEL
LIN {X 0,Y 473.723,Z 404.048,A -85,B 0,C 180,E1 -7292.55,E2 -7292.55} C_VEL
LIN {X 0,Y 473.765,Z 402.646,A -85,B 0,C 180,E1 -7293.401,E2 -7293.401} C_VEL
LIN {X 0,Y 473.762,Z 399.698,A -85,B 0,C 180,E1 -7294.679,E2 -7294.679} C_VEL
LIN {X 0,Y 473.864,Z 395.708,A -85,B 0,C 180,E1 -7295.958,E2 -7295.958} C_VEL
LIN {X 0,Y 474.029,Z 389.57,A -85,B 0,C 180,E1 -7297.453,E2 -7297.453} C_VEL
LIN {X 0,Y 474.297,Z 382.865,A -85,B 0,C 180,E1 -7298.735,E2 -7298.735} C_VEL
LIN {X 0,Y 474.648,Z 374.546,A -85,B 0,C 180,E1 -7300.018,E2 -7300.018} C_VEL
LIN {X 0,Y 475.034,Z 366.003,A -85,B 0,C 180,E1 -7301.088,E2 -7301.088} C_VEL
LIN {X 0,Y 475.51,Z 355.545,A -85,B 0,C 180,E1 -7302.149,E2 -7302.149} C_VEL
LIN {X 0,Y 475.973,Z 343.718,A -85,B 0,C 180,E1 -7303.109,E2 -7303.109} C_VEL
LIN {X 0,Y 476.413,Z 331.56,A -85,B 0,C 180,E1 -7303.869,E2 -7303.869} C_VEL
LIN {X 0,Y 476.938,Z 319.071,A -85,B 0,C 180,E1 -7304.452,E2 -7304.452} C_VEL
LIN {X 0,Y 477.253,Z 306.073,A -85,B 0,C 180,E1 -7304.878,E2 -7304.878} C_VEL
LIN {X 0,Y 477.498,Z 290.521,A -85,B 0,C 180,E1 -7305.17,E2 -7305.17} C_VEL
LIN {X 0,Y 477.956,Z 209.756,A -85,B 0,C 180,E1 -7306.427,E2 -7306.427} C_VEL
LIN {X 0,Y 475.415,Z 194.114,A -85,B 0,C 180,E1 -7306.78,E2 -7306.78} C_VEL
LIN {X 0,Y 475.396,Z 192.586,A -85,B 0,C 180,E1 -7306.975,E2 -7306.975} C_VEL
LIN {X 0,Y 475.998,Z 175.375,A -85,B 0,C 180,E1 -7310.076,E2 -7310.076} C_VEL
LIN {X 0,Y 476.534,Z 161.862,A -85,B 0,C 180,E1 -7312.546,E2 -7312.546} C_VEL
LIN {X 0,Y 474.855,Z 152.014,A -85,B 0,C 180,E1 -7314.481,E2 -7314.481} C_VEL
LIN {X 0,Y 474.633,Z 150.893,A -85,B 0,C 180,E1 -7314.785,E2 -7314.785} C_VEL
LIN {X 0,Y 474.585,Z 150.869,A -85,B 0,C 180,E1 -7318.285,E2 -7318.285} C_VEL
LIN {X 0,Y 474.573,Z 150.87,A -85,B 0,C 180,E1 -7321.218,E2 -7321.218} C_VEL
LIN {X 0,Y 474.612,Z 150.864,A -85,B 0,C 180,E1 -7324.241,E2 -7324.241} C_VEL
LIN {X 0,Y 474.531,Z 150.879,A -85,B 0,C 180,E1 -7327.387,E2 -7327.387} C_VEL
LIN {X 0,Y 474.591,Z 150.869,A -85,B 0,C 180,E1 -7329.642,E2 -7329.642} C_VEL
LIN {X 0,Y 474.567,Z 150.868,A -85,B 0,C 180,E1 -7332.229,E2 -7332.229} C_VEL
LIN {X 0,Y 474.604,Z 150.87,A -85,B 0,C 180,E1 -7335.297,E2 -7335.297} C_VEL
LIN {X 0,Y 474.582,Z 150.866,A -85,B 0,C 180,E1 -7338.21,E2 -7338.21} C_VEL
LIN {X 0,Y 474.59,Z 150.866,A -85,B 0,C 180,E1 -7341.54,E2 -7341.54} C_VEL
LIN {X 0,Y 474.608,Z 150.865,A -85,B 0,C 180,E1 -7344.724,E2 -7344.724} C_VEL
LIN {X 0,Y 474.605,Z 150.862,A -85,B 0,C 180,E1 -7347.785,E2 -7347.785} C_VEL
LIN {X 0,Y 474.582,Z 150.871,A -85,B 0,C 180,E1 -7350.89,E2 -7350.89} C_VEL
LIN {X 0,Y 474.57,Z 150.867,A -85,B 0,C 180,E1 -7353.623,E2 -7353.623} C_VEL
LIN {X 0,Y 474.622,Z 150.863,A -85,B 0,C 180,E1 -7356.641,E2 -7356.641} C_VEL
LIN {X 0,Y 474.637,Z 150.857,A -85,B 0,C 180,E1 -7360.088,E2 -7360.088} C_VEL
LIN {X 0,Y 474.619,Z 150.866,A -85,B 0,C 180,E1 -7362.773,E2 -7362.773} C_VEL
